LIN {X 0,Y 466.003,Z 780.81,A -85,B 0,C 180,E1 14179.349,E2 14179.349} C_VEL
LIN {X 0,Y 466.055,Z 780.81,A -85,B 0,C 180,E1 14186.554,E2 14186.554} C_VEL
LIN {X 0,Y 466.342,Z 780.81,A -85,B 0,C 180,E1 14193.024,E2 14193.024} C_VEL
LIN {X 0,Y 466.575,Z 780.81,A -85,B 0,C 180,E1 14199.925,E2 14199.925} C_VEL
LIN {X 0,Y 466.793,Z 780.81,A -85,B 0,C 180,E1 14206.211,E2 14206.211} C_VEL
LIN {X 0,Y 467.178,Z 780.81,A -85,B 0,C 180,E1 14212.565,E2 14212.565} C_VEL
LIN {X 0,Y 467.507,Z 780.81,A -85,B 0,C 180,E1 14218.145,E2 14218.145} C_VEL
LIN {X 0,Y 467.363,Z 780.81,A -85,B 0,C 180,E1 14223.704,E2 14223.704} C_VEL
LIN {X 0,Y 467.109,Z 780.81,A -85,B 0,C 180,E1 14229.304,E2 14229.304} C_VEL
LIN {X 0,Y 466.805,Z 780.81,A -85,B 0,C 180,E1 14235.003,E2 14235.003} C_VEL
LIN {X 0,Y 466.56,Z 780.81,A -85,B 0,C 180,E1 14240.865,E2 14240.865} C_VEL
LIN {X 0,Y 466.356,Z 780.81,A -85,B 0,C 180,E1 14246.969,E2 14246.969} C_VEL
LIN {X 0,Y 466.141,Z 780.81,A -85,B 0,C 180,E1 14253.432,E2 14253.432} C_VEL
LIN {X 0,Y 466.096,Z 780.943,A -85,B 0,C 180,E1 14257.269,E2 14257.269} C_VEL
LIN {X 0,Y 468.35,Z 786.358,A -85,B 0,C 180,E1 14257.738,E2 14257.738} C_VEL
LIN {X 0,Y 490.215,Z 820.764,A -85,B 0,C 180,E1 14261.492,E2 14261.492} C_VEL
LIN {X 0,Y 509.708,Z 858.555,A -85,B 0,C 180,E1 14264.767,E2 14264.767} C_VEL
LIN {X 0,Y 518.237,Z 880.593,A -85,B 0,C 180,E1 14266.483,E2 14266.483} C_VEL
LIN {X 0,Y 512.004,Z 925.358,A -85,B 0,C 180,E1 14268.177,E2 14268.177} C_VEL
LIN {X 0,Y 504.346,Z 968.699,A -85,B 0,C 180,E1 14270.608,E2 14270.608} C_VEL
LIN {X 0,Y 495.859,Z 1008.879,A -85,B 0,C 180,E1 14273.729,E2 14273.729} C_VEL
LIN {X 0,Y 487.965,Z 1043.053,A -85,B 0,C 180,E1 14277.25,E2 14277.25} C_VEL
LIN {X 0,Y 480.836,Z 1073.807,A -85,B 0,C 180,E1 14281.363,E2 14281.363} C_VEL
LIN {X 0,Y 474.612,Z 1101.899,A -85,B 0,C 180,E1 14286.298,E2 14286.298} C_VEL
LIN {X 0,Y 470.527,Z 1124.762,A -85,B 0,C 180,E1 14291.751,E2 14291.751} C_VEL
LIN {X 0,Y 468.531,Z 1140.188,A -85,B 0,C 180,E1 14296.951,E2 14296.951} C_VEL
LIN {X 0,Y 467.871,Z 1149.631,A -85,B 0,C 180,E1 14301.642,E2 14301.642} C_VEL
LIN {X 0,Y 467.662,Z 1154.817,A -85,B 0,C 180,E1 14306.294,E2 14306.294} C_VEL
LIN {X 0,Y 467.72,Z 1156.159,A -85,B 0,C 180,E1 14309.999,E2 14309.999} C_VEL
LIN {X 0,Y 467.629,Z 1155.649,A -85,B 0,C 180,E1 14312.192,E2 14312.192} C_VEL
LIN {X 0,Y 463.625,Z 1154.407,A -85,B 0,C 180,E1 14314.275,E2 14314.275} C_VEL
LIN {X 0,Y 459.843,Z 1152.277,A -85,B 0,C 180,E1 14316.387,E2 14316.387} C_VEL
LIN {X 0,Y 460.346,Z 1144.47,A -85,B 0,C 180,E1 14321.358,E2 14321.358} C_VEL
LIN {X 0,Y 461.991,Z 1131.343,A -85,B 0,C 180,E1 14326.629,E2 14326.629} C_VEL
LIN {X 0,Y 465.491,Z 1111.513,A -85,B 0,C 180,E1 14332.135,E2 14332.135} C_VEL
LIN {X 0,Y 471.08,Z 1086.781,A -85,B 0,C 180,E1 14337.199,E2 14337.199} C_VEL
LIN {X 0,Y 478.526,Z 1057.544,A -85,B 0,C 180,E1 14341.738,E2 14341.738} C_VEL
LIN {X 0,Y 487.44,Z 1023.022,A -85,B 0,C 180,E1 14345.812,E2 14345.812} C_VEL
LIN {X 0,Y 497.158,Z 982.841,A -85,B 0,C 180,E1 14349.34,E2 14349.34} C_VEL
LIN {X 0,Y 506.149,Z 940.056,A -85,B 0,C 180,E1 14352.054,E2 14352.054} C_VEL
LIN {X 0,Y 513.496,Z 896.79,A -85,B 0,C 180,E1 14353.955,E2 14353.955} C_VEL
LIN {X 0,Y 514.956,Z 882.197,A -85,B 0,C 180,E1 14354.501,E2 14354.501} C_VEL
LIN {X 0,Y 499.256,Z 847.046,A -85,B 0,C 180,E1 14357.774,E2 14357.774} C_VEL
LIN {X 0,Y 478.485,Z 812.037,A -85,B 0,C 180,E1 14361.711,E2 14361.711} C_VEL
LIN {X 0,Y 464.229,Z 791.641,A -85,B 0,C 180,E1 14364.642,E2 14364.642} C_VEL
LIN {X 0,Y 461.04,Z 786.903,A -85,B 0,C 180,E1 14365.359,E2 14365.359} C_VEL
LIN {X 0,Y 458.257,Z 781.978,A -85,B 0,C 180,E1 14366.028,E2 14366.028} C_VEL
LIN {X 0,Y 458.165,Z 780.81,A -85,B 0,C 180,E1 14366.133,E2 14366.133} C_VEL
LIN {X 0,Y 458.415,Z 780.81,A -85,B 0,C 180,E1 14372.873,E2 14372.873} C_VEL
LIN {X 0,Y 458.576,Z 780.81,A -85,B 0,C 180,E1 14378.755,E2 14378.755} C_VEL
LIN {X 0,Y 458.834,Z 780.81,A -85,B 0,C 180,E1 14384.73,E2 14384.73} C_VEL
LIN {X 0,Y 459.194,Z 780.81,A -85,B 0,C 180,E1 14390.828,E2 14390.828} C_VEL
LIN {X 0,Y 459.536,Z 780.81,A -85,B 0,C 180,E1 14396.233,E2 14396.233} C_VEL
LIN {X 0,Y 459.624,Z 780.81,A -85,B 0,C 180,E1 14401.887,E2 14401.887} C_VEL
LIN {X 0,Y 459.276,Z 780.81,A -85,B 0,C 180,E1 14407.564,E2 14407.564} C_VEL
LIN {X 0,Y 459.011,Z 780.81,A -85,B 0,C 180,E1 14413.324,E2 14413.324} C_VEL
LIN {X 0,Y 458.683,Z 780.81,A -85,B 0,C 180,E1 14419.235,E2 14419.235} C_VEL
LIN {X 0,Y 458.385,Z 780.81,A -85,B 0,C 180,E1 14425.374,E2 14425.374} C_VEL
LIN {X 0,Y 458.219,Z 780.81,A -85,B 0,C 180,E1 14431.37,E2 14431.37} C_VEL
LIN {X 0,Y 460.406,Z 786.283,A -85,B 0,C 180,E1 14431.966,E2 14431.966} C_VEL
LIN {X 0,Y 463.2,Z 789.773,A -85,B 0,C 180,E1 14432.582,E2 14432.582} C_VEL
LIN {X 0,Y 482.614,Z 818.941,A -85,B 0,C 180,E1 14436.642,E2 14436.642} C_VEL
LIN {X 0,Y 500.16,Z 852.088,A -85,B 0,C 180,E1 14440.434,E2 14440.434} C_VEL
LIN {X 0,Y 512.562,Z 884.16,A -85,B 0,C 180,E1 14443.642,E2 14443.642} C_VEL
LIN {X 0,Y 504.897,Z 927.615,A -85,B 0,C 180,E1 14445.867,E2 14445.867} C_VEL
LIN {X 0,Y 496.016,Z 968.133,A -85,B 0,C 180,E1 14448.793,E2 14448.793} C_VEL
LIN {X 0,Y 486.772,Z 1004.454,A -85,B 0,C 180,E1 14452.331,E2 14452.331} C_VEL
LIN {X 0,Y 478.378,Z 1035.552,A -85,B 0,C 180,E1 14456.331,E2 14456.331} C_VEL
LIN {X 0,Y 471.191,Z 1062.29,A -85,B 0,C 180,E1 14460.815,E2 14460.815} C_VEL
LIN {X 0,Y 465.51,Z 1085.609,A -85,B 0,C 180,E1 14466.062,E2 14466.062} C_VEL
LIN {X 0,Y 462.178,Z 1102.875,A -85,B 0,C 180,E1 14471.451,E2 14471.451} C_VEL
LIN {X 0,Y 460.451,Z 1114.458,A -85,B 0,C 180,E1 14476.72,E2 14476.72} C_VEL
LIN {X 0,Y 459.92,Z 1119.813,A -85,B 0,C 180,E1 14480.546,E2 14480.546} C_VEL
LIN {X 0,Y 459.641,Z 1123.056,A -85,B 0,C 180,E1 14486.231,E2 14486.231} C_VEL
LIN {X 0,Y 459.933,Z 1120.944,A -85,B 0,C 180,E1 14491.884,E2 14491.884} C_VEL
LIN {X 0,Y 460.385,Z 1115.045,A -85,B 0,C 180,E1 14496.598,E2 14496.598} C_VEL
LIN {X 0,Y 461.817,Z 1103.979,A -85,B 0,C 180,E1 14501.802,E2 14501.802} C_VEL
LIN {X 0,Y 464.72,Z 1087.594,A -85,B 0,C 180,E1 14507.018,E2 14507.018} C_VEL
LIN {X 0,Y 469.803,Z 1064.997,A -85,B 0,C 180,E1 14512.207,E2 14512.207} C_VEL
LIN {X 0,Y 476.391,Z 1038.632,A -85,B 0,C 180,E1 14516.752,E2 14516.752} C_VEL
LIN {X 0,Y 484.526,Z 1006.922,A -85,B 0,C 180,E1 14520.912,E2 14520.912} C_VEL
LIN {X 0,Y 493.645,Z 968.867,A -85,B 0,C 180,E1 14524.653,E2 14524.653} C_VEL
LIN {X 0,Y 502.271,Z 927.064,A -85,B 0,C 180,E1 14527.671,E2 14527.671} C_VEL
LIN {X 0,Y 509.568,Z 883.42,A -85,B 0,C 180,E1 14529.892,E2 14529.892} C_VEL
LIN {X 0,Y 495.699,Z 847.197,A -85,B 0,C 180,E1 14533.224,E2 14533.224} C_VEL
LIN {X 0,Y 476.674,Z 811.093,A -85,B 0,C 180,E1 14536.915,E2 14536.915} C_VEL
LIN {X 0,Y 460.205,Z 786.237,A -85,B 0,C 180,E1 14539.979,E2 14539.979} C_VEL
LIN {X 0,Y 458.009,Z 780.81,A -85,B 0,C 180,E1 14540.535,E2 14540.535} C_VEL
LIN {X 0,Y 458.055,Z 780.81,A -85,B 0,C 180,E1 14545.89,E2 14545.89} C_VEL
LIN {X 0,Y 458.379,Z 780.81,A -85,B 0,C 180,E1 14552.516,E2 14552.516} C_VEL
LIN {X 0,Y 458.588,Z 780.81,A -85,B 0,C 180,E1 14558.749,E2 14558.749} C_VEL
LIN {X 0,Y 458.832,Z 780.81,A -85,B 0,C 180,E1 14564.724,E2 14564.724} C_VEL
LIN {X 0,Y 459.215,Z 780.81,A -85,B 0,C 180,E1 14570.825,E2 14570.825} C_VEL
LIN {X 0,Y 459.558,Z 780.81,A -85,B 0,C 180,E1 14576.227,E2 14576.227} C_VEL
LIN {X 0,Y 459.639,Z 780.81,A -85,B 0,C 180,E1 14581.881,E2 14581.881} C_VEL
LIN {X 0,Y 459.248,Z 780.81,A -85,B 0,C 180,E1 14587.559,E2 14587.559} C_VEL
LIN {X 0,Y 458.996,Z 780.81,A -85,B 0,C 180,E1 14593.319,E2 14593.319} C_VEL
LIN {X 0,Y 458.715,Z 780.81,A -85,B 0,C 180,E1 14599.227,E2 14599.227} C_VEL
LIN {X 0,Y 458.424,Z 780.81,A -85,B 0,C 180,E1 14605.366,E2 14605.366} C_VEL
LIN {X 0,Y 458.26,Z 780.81,A -85,B 0,C 180,E1 14611.834,E2 14611.834} C_VEL
LIN {X 0,Y 458.148,Z 781.129,A -85,B 0,C 180,E1 14616.023,E2 14616.023} C_VEL
LIN {X 0,Y 460.626,Z 786.52,A -85,B 0,C 180,E1 14616.555,E2 14616.555} C_VEL
LIN {X 0,Y 480.891,Z 818.052,A -85,B 0,C 180,E1 14620.229,E2 14620.229} C_VEL
LIN {X 0,Y 500.554,Z 854.498,A -85,B 0,C 180,E1 14623.632,E2 14623.632} C_VEL
LIN {X 0,Y 512.078,Z 882.629,A -85,B 0,C 180,E1 14625.954,E2 14625.954} C_VEL
LIN {X 0,Y 505.842,Z 925.769,A -85,B 0,C 180,E1 14627.621,E2 14627.621} C_VEL
LIN {X 0,Y 497.732,Z 969.89,A -85,B 0,C 180,E1 14630.137,E2 14630.137} C_VEL
LIN {X 0,Y 488.886,Z 1010.227,A -85,B 0,C 180,E1 14633.327,E2 14633.327} C_VEL
LIN {X 0,Y 480.144,Z 1046.596,A -85,B 0,C 180,E1 14637.199,E2 14637.199} C_VEL
LIN {X 0,Y 472.886,Z 1076.357,A -85,B 0,C 180,E1 14641.358,E2 14641.358} C_VEL
LIN {X 0,Y 466.88,Z 1102.629,A -85,B 0,C 180,E1 14646.134,E2 14646.134} C_VEL
LIN {X 0,Y 462.745,Z 1124.874,A -85,B 0,C 180,E1 14651.571,E2 14651.571} C_VEL
LIN {X 0,Y 460.587,Z 1141.036,A -85,B 0,C 180,E1 14657.204,E2 14657.204} C_VEL
LIN {X 0,Y 459.892,Z 1150.634,A -85,B 0,C 180,E1 14662.447,E2 14662.447} C_VEL
LIN {X 0,Y 459.836,Z 1155.529,A -85,B 0,C 180,E1 14668.116,E2 14668.116} C_VEL
LIN {X 0,Y 459.733,Z 1155.398,A -85,B 0,C 180,E1 14672.175,E2 14672.175} C_VEL
LIN {X 0,Y 459.843,Z 1152.277,A -85,B 0,C 180,E1 14676.387,E2 14676.387} C_VEL
LIN {X 0,Y 457.472,Z 1150.386,A -85,B 0,C 180,E1 14677.982,E2 14677.982} C_VEL
LIN {X 0,Y 452.366,Z 1146.556,A -85,B 0,C 180,E1 14680.355,E2 14680.355} C_VEL
LIN {X 0,Y 452.306,Z 1146.036,A -85,B 0,C 180,E1 14680.627,E2 14680.627} C_VEL
LIN {X 0,Y 453.777,Z 1133.828,A -85,B 0,C 180,E1 14685.945,E2 14685.945} C_VEL
LIN {X 0,Y 456.962,Z 1116.098,A -85,B 0,C 180,E1 14691.33,E2 14691.33} C_VEL
LIN {X 0,Y 462.798,Z 1090.841,A -85,B 0,C 180,E1 14696.893,E2 14696.893} C_VEL
LIN {X 0,Y 470.93,Z 1060.042,A -85,B 0,C 180,E1 14701.903,E2 14701.903} C_VEL
LIN {X 0,Y 480.579,Z 1024.039,A -85,B 0,C 180,E1 14706.264,E2 14706.264} C_VEL
LIN {X 0,Y 490.627,Z 984.162,A -85,B 0,C 180,E1 14709.83,E2 14709.83} C_VEL
LIN {X 0,Y 499.865,Z 941.995,A -85,B 0,C 180,E1 14712.562,E2 14712.562} C_VEL
LIN {X 0,Y 507.349,Z 900.29,A -85,B 0,C 180,E1 14714.452,E2 14714.452} C_VEL
LIN {X 0,Y 508.891,Z 884.922,A -85,B 0,C 180,E1 14715.065,E2 14715.065} C_VEL
LIN {X 0,Y 493.722,Z 850.498,A -85,B 0,C 180,E1 14718.391,E2 14718.391} C_VEL
LIN {X 0,Y 474.535,Z 817.647,A -85,B 0,C 180,E1 14722.205,E2 14722.205} C_VEL
LIN {X 0,Y 457.343,Z 792.903,A -85,B 0,C 180,E1 14725.895,E2 14725.895} C_VEL
LIN {X 0,Y 453.216,Z 786.958,A -85,B 0,C 180,E1 14726.882,E2 14726.882} C_VEL
LIN {X 0,Y 450.415,Z 782.207,A -85,B 0,C 180,E1 14727.6,E2 14727.6} C_VEL
LIN {X 0,Y 450.283,Z 780.81,A -85,B 0,C 180,E1 14727.756,E2 14727.756} C_VEL
LIN {X 0,Y 450.496,Z 780.81,A -85,B 0,C 180,E1 14734.155,E2 14734.155} C_VEL
LIN {X 0,Y 450.716,Z 780.81,A -85,B 0,C 180,E1 14740.418,E2 14740.418} C_VEL
LIN {X 0,Y 451.016,Z 780.81,A -85,B 0,C 180,E1 14746.441,E2 14746.441} C_VEL
LIN {X 0,Y 451.316,Z 780.81,A -85,B 0,C 180,E1 14752.308,E2 14752.308} C_VEL
LIN {X 0,Y 451.682,Z 780.81,A -85,B 0,C 180,E1 14758.086,E2 14758.086} C_VEL
LIN {X 0,Y 451.543,Z 780.81,A -85,B 0,C 180,E1 14763.84,E2 14763.84} C_VEL
LIN {X 0,Y 451.271,Z 780.81,A -85,B 0,C 180,E1 14769.64,E2 14769.64} C_VEL
LIN {X 0,Y 450.963,Z 780.81,A -85,B 0,C 180,E1 14775.55,E2 14775.55} C_VEL
LIN {X 0,Y 450.632,Z 780.81,A -85,B 0,C 180,E1 14781.645,E2 14781.645} C_VEL
LIN {X 0,Y 450.369,Z 780.81,A -85,B 0,C 180,E1 14788.015,E2 14788.015} C_VEL
LIN {X 0,Y 450.369,Z 781.276,A -85,B 0,C 180,E1 14789.825,E2 14789.825} C_VEL
LIN {X 0,Y 452.709,Z 786.471,A -85,B 0,C 180,E1 14790.463,E2 14790.463} C_VEL
LIN {X 0,Y 455.413,Z 789.825,A -85,B 0,C 180,E1 14791.103,E2 14791.103} C_VEL
LIN {X 0,Y 472.547,Z 815.076,A -85,B 0,C 180,E1 14794.929,E2 14794.929} C_VEL
LIN {X 0,Y 489.417,Z 844.882,A -85,B 0,C 180,E1 14798.666,E2 14798.666} C_VEL
LIN {X 0,Y 503.111,Z 877.093,A -85,B 0,C 180,E1 14802.12,E2 14802.12} C_VEL
LIN {X 0,Y 506.394,Z 888.401,A -85,B 0,C 180,E1 14803.199,E2 14803.199} C_VEL
LIN {X 0,Y 498.875,Z 928.512,A -85,B 0,C 180,E1 14805.288,E2 14805.288} C_VEL
LIN {X 0,Y 489.595,Z 969.436,A -85,B 0,C 180,E1 14808.28,E2 14808.28} C_VEL
LIN {X 0,Y 479.894,Z 1006.088,A -85,B 0,C 180,E1 14811.917,E2 14811.917} C_VEL
LIN {X 0,Y 471.205,Z 1036.913,A -85,B 0,C 180,E1 14815.973,E2 14815.973} C_VEL
LIN {X 0,Y 463.985,Z 1062.615,A -85,B 0,C 180,E1 14820.363,E2 14820.363} C_VEL
LIN {X 0,Y 457.973,Z 1086.049,A -85,B 0,C 180,E1 14825.721,E2 14825.721} C_VEL
LIN {X 0,Y 454.402,Z 1103.478,A -85,B 0,C 180,E1 14831.279,E2 14831.279} C_VEL
LIN {X 0,Y 452.616,Z 1114.687,A -85,B 0,C 180,E1 14836.486,E2 14836.486} C_VEL
LIN {X 0,Y 451.835,Z 1121.751,A -85,B 0,C 180,E1 14842.313,E2 14842.313} C_VEL
LIN {X 0,Y 451.783,Z 1123.23,A -85,B 0,C 180,E1 14848.084,E2 14848.084} C_VEL
LIN {X 0,Y 452.171,Z 1119.382,A -85,B 0,C 180,E1 14853.833,E2 14853.833} C_VEL
LIN {X 0,Y 453.146,Z 1110.057,A -85,B 0,C 180,E1 14859.599,E2 14859.599} C_VEL
LIN {X 0,Y 455.801,Z 1094.608,A -85,B 0,C 180,E1 14865.381,E2 14865.381} C_VEL
LIN {X 0,Y 460.243,Z 1074.335,A -85,B 0,C 180,E1 14870.689,E2 14870.689} C_VEL
LIN {X 0,Y 466.4,Z 1050.103,A -85,B 0,C 180,E1 14875.424,E2 14875.424} C_VEL
LIN {X 0,Y 474.359,Z 1020.232,A -85,B 0,C 180,E1 14879.852,E2 14879.852} C_VEL
LIN {X 0,Y 483.758,Z 983.33,A -85,B 0,C 180,E1 14883.943,E2 14883.943} C_VEL
LIN {X 0,Y 493.261,Z 942.016,A -85,B 0,C 180,E1 14887.293,E2 14887.293} C_VEL
LIN {X 0,Y 501.024,Z 901.017,A -85,B 0,C 180,E1 14889.687,E2 14889.687} C_VEL
LIN {X 0,Y 503.111,Z 885.592,A -85,B 0,C 180,E1 14890.437,E2 14890.437} C_VEL
LIN {X 0,Y 489.101,Z 848.95,A -85,B 0,C 180,E1 14893.943,E2 14893.943} C_VEL
LIN {X 0,Y 471.255,Z 814.96,A -85,B 0,C 180,E1 14897.571,E2 14897.571} C_VEL
LIN {X 0,Y 452.843,Z 786.776,A -85,B 0,C 180,E1 14901.17,E2 14901.17} C_VEL
LIN {X 0,Y 450.18,Z 782.05,A -85,B 0,C 180,E1 14901.749,E2 14901.749} C_VEL
LIN {X 0,Y 450.107,Z 780.81,A -85,B 0,C 180,E1 14901.897,E2 14901.897} C_VEL
LIN {X 0,Y 450.174,Z 780.81,A -85,B 0,C 180,E1 14907.518,E2 14907.518} C_VEL
LIN {X 0,Y 450.47,Z 780.81,A -85,B 0,C 180,E1 14914.147,E2 14914.147} C_VEL
LIN {X 0,Y 450.728,Z 780.81,A -85,B 0,C 180,E1 14920.412,E2 14920.412} C_VEL
LIN {X 0,Y 451.015,Z 780.81,A -85,B 0,C 180,E1 14926.435,E2 14926.435} C_VEL
LIN {X 0,Y 451.327,Z 780.81,A -85,B 0,C 180,E1 14933.141,E2 14933.141} C_VEL
LIN {X 0,Y 451.713,Z 780.81,A -85,B 0,C 180,E1 14938.08,E2 14938.08} C_VEL
LIN {X 0,Y 451.541,Z 780.81,A -85,B 0,C 180,E1 14943.834,E2 14943.834} C_VEL
LIN {X 0,Y 451.26,Z 780.81,A -85,B 0,C 180,E1 14949.634,E2 14949.634} C_VEL
LIN {X 0,Y 450.932,Z 780.81,A -85,B 0,C 180,E1 14955.545,E2 14955.545} C_VEL
LIN {X 0,Y 450.661,Z 780.81,A -85,B 0,C 180,E1 14961.637,E2 14961.637} C_VEL
LIN {X 0,Y 450.406,Z 780.81,A -85,B 0,C 180,E1 14968.006,E2 14968.006} C_VEL
LIN {X 0,Y 450.224,Z 780.81,A -85,B 0,C 180,E1 14974.66,E2 14974.66} C_VEL
LIN {X 0,Y 452.498,Z 786.331,A -85,B 0,C 180,E1 14975.221,E2 14975.221} C_VEL
LIN {X 0,Y 468.108,Z 809.74,A -85,B 0,C 180,E1 14978.254,E2 14978.254} C_VEL
LIN {X 0,Y 488.269,Z 844.522,A -85,B 0,C 180,E1 14981.862,E2 14981.862} C_VEL
LIN {X 0,Y 504.735,Z 881.742,A -85,B 0,C 180,E1 14985.154,E2 14985.154} C_VEL
LIN {X 0,Y 505.776,Z 886.831,A -85,B 0,C 180,E1 14985.49,E2 14985.49} C_VEL
LIN {X 0,Y 499.132,Z 929.42,A -85,B 0,C 180,E1 14987.211,E2 14987.211} C_VEL
LIN {X 0,Y 491.175,Z 970.88,A -85,B 0,C 180,E1 14989.64,E2 14989.64} C_VEL
LIN {X 0,Y 482.094,Z 1010.81,A -85,B 0,C 180,E1 14992.848,E2 14992.848} C_VEL
LIN {X 0,Y 472.801,Z 1048.094,A -85,B 0,C 180,E1 14996.898,E2 14996.898} C_VEL
LIN {X 0,Y 464.517,Z 1080.856,A -85,B 0,C 180,E1 15001.671,E2 15001.671} C_VEL
LIN {X 0,Y 458.291,Z 1107.776,A -85,B 0,C 180,E1 15006.943,E2 15006.943} C_VEL
LIN {X 0,Y 454.536,Z 1127.489,A -85,B 0,C 180,E1 15012.173,E2 15012.173} C_VEL
LIN {X 0,Y 452.637,Z 1141.837,A -85,B 0,C 180,E1 15017.466,E2 15017.466} C_VEL
LIN {X 0,Y 452.023,Z 1150.33,A -85,B 0,C 180,E1 15022.314,E2 15022.314} C_VEL
LIN {X 0,Y 451.955,Z 1155.246,A -85,B 0,C 180,E1 15028.083,E2 15028.083} C_VEL
LIN {X 0,Y 451.902,Z 1155.269,A -85,B 0,C 180,E1 15031.915,E2 15031.915} C_VEL
LIN {X 0,Y 452.025,Z 1150.557,A -85,B 0,C 180,E1 15037.683,E2 15037.683} C_VEL
LIN {X 0,Y 452.306,Z 1146.036,A -85,B 0,C 180,E1 15040.627,E2 15040.627} C_VEL
LIN {X 0,Y 448.774,Z 1141.925,A -85,B 0,C 180,E1 15042.743,E2 15042.743} C_VEL
LIN {X 0,Y 445.465,Z 1137.142,A -85,B 0,C 180,E1 15044.878,E2 15044.878} C_VEL
LIN {X 0,Y 448.218,Z 1121.269,A -85,B 0,C 180,E1 15050.215,E2 15050.215} C_VEL
LIN {X 0,Y 453.373,Z 1098.991,A -85,B 0,C 180,E1 15055.675,E2 15055.675} C_VEL
LIN {X 0,Y 461.021,Z 1070.776,A -85,B 0,C 180,E1 15060.806,E2 15060.806} C_VEL
LIN {X 0,Y 470.809,Z 1035.517,A -85,B 0,C 180,E1 15065.572,E2 15065.572} C_VEL
LIN {X 0,Y 481.48,Z 996.197,A -85,B 0,C 180,E1 15069.466,E2 15069.466} C_VEL
LIN {X 0,Y 491.726,Z 953.378,A -85,B 0,C 180,E1 15072.536,E2 15072.536} C_VEL
LIN {X 0,Y 499.965,Z 911.064,A -85,B 0,C 180,E1 15074.671,E2 15074.671} C_VEL
LIN {X 0,Y 502.984,Z 887.991,A -85,B 0,C 180,E1 15075.613,E2 15075.613} C_VEL
LIN {X 0,Y 488.697,Z 854.787,A -85,B 0,C 180,E1 15078.931,E2 15078.931} C_VEL
LIN {X 0,Y 470.369,Z 822.869,A -85,B 0,C 180,E1 15082.755,E2 15082.755} C_VEL
LIN {X 0,Y 453.676,Z 798.649,A -85,B 0,C 180,E1 15086.449,E2 15086.449} C_VEL
LIN {X 0,Y 445.848,Z 787.309,A -85,B 0,C 180,E1 15088.421,E2 15088.421} C_VEL
LIN {X 0,Y 442.676,Z 782.833,A -85,B 0,C 180,E1 15089.271,E2 15089.271} C_VEL
LIN {X 0,Y 442.415,Z 780.81,A -85,B 0,C 180,E1 15089.433,E2 15089.433} C_VEL
LIN {X 0,Y 442.587,Z 780.81,A -85,B 0,C 180,E1 15095.821,E2 15095.821} C_VEL
LIN {X 0,Y 442.923,Z 780.81,A -85,B 0,C 180,E1 15102.794,E2 15102.794} C_VEL
LIN {X 0,Y 443.167,Z 780.81,A -85,B 0,C 180,E1 15108.2,E2 15108.2} C_VEL
LIN {X 0,Y 443.508,Z 780.81,A -85,B 0,C 180,E1 15114.137,E2 15114.137} C_VEL
LIN {X 0,Y 443.961,Z 780.81,A -85,B 0,C 180,E1 15120.003,E2 15120.003} C_VEL
LIN {X 0,Y 443.58,Z 780.81,A -85,B 0,C 180,E1 15125.868,E2 15125.868} C_VEL
LIN {X 0,Y 443.208,Z 780.81,A -85,B 0,C 180,E1 15131.805,E2 15131.805} C_VEL
LIN {X 0,Y 442.903,Z 780.81,A -85,B 0,C 180,E1 15137.882,E2 15137.882} C_VEL
LIN {X 0,Y 442.562,Z 780.81,A -85,B 0,C 180,E1 15144.187,E2 15144.187} C_VEL
LIN {X 0,Y 442.467,Z 780.935,A -85,B 0,C 180,E1 15148.083,E2 15148.083} C_VEL
LIN {X 0,Y 444.419,Z 786.044,A -85,B 0,C 180,E1 15148.687,E2 15148.687} C_VEL
LIN {X 0,Y 447.508,Z 789.498,A -85,B 0,C 180,E1 15149.469,E2 15149.469} C_VEL
LIN {X 0,Y 465.321,Z 815.546,A -85,B 0,C 180,E1 15153.715,E2 15153.715} C_VEL
LIN {X 0,Y 482.559,Z 845.746,A -85,B 0,C 180,E1 15157.721,E2 15157.721} C_VEL
LIN {X 0,Y 496.416,Z 878.028,A -85,B 0,C 180,E1 15161.345,E2 15161.345} C_VEL
LIN {X 0,Y 500.471,Z 890.799,A -85,B 0,C 180,E1 15162.652,E2 15162.652} C_VEL
LIN {X 0,Y 492.587,Z 930.897,A -85,B 0,C 180,E1 15164.792,E2 15164.792} C_VEL
LIN {X 0,Y 483.194,Z 970.718,A -85,B 0,C 180,E1 15167.755,E2 15167.755} C_VEL
LIN {X 0,Y 473.022,Z 1007.812,A -85,B 0,C 180,E1 15171.502,E2 15171.502} C_VEL
LIN {X 0,Y 463.69,Z 1039.531,A -85,B 0,C 180,E1 15175.796,E2 15175.796} C_VEL
LIN {X 0,Y 455.858,Z 1066.093,A -85,B 0,C 180,E1 15180.551,E2 15180.551} C_VEL
LIN {X 0,Y 450.004,Z 1088.196,A -85,B 0,C 180,E1 15185.847,E2 15185.847} C_VEL
LIN {X 0,Y 446.324,Z 1105.875,A -85,B 0,C 180,E1 15191.798,E2 15191.798} C_VEL
LIN {X 0,Y 444.603,Z 1116.444,A -85,B 0,C 180,E1 15197.238,E2 15197.238} C_VEL
LIN {X 0,Y 443.943,Z 1122.004,A -85,B 0,C 180,E1 15202.176,E2 15202.176} C_VEL
LIN {X 0,Y 443.883,Z 1123.517,A -85,B 0,C 180,E1 15208.05,E2 15208.05} C_VEL
LIN {X 0,Y 444.284,Z 1119.706,A -85,B 0,C 180,E1 15213.902,E2 15213.902} C_VEL
LIN {X 0,Y 445.315,Z 1110.413,A -85,B 0,C 180,E1 15219.77,E2 15219.77} C_VEL
LIN {X 0,Y 448.115,Z 1094.999,A -85,B 0,C 180,E1 15225.652,E2 15225.652} C_VEL
LIN {X 0,Y 452.757,Z 1074.82,A -85,B 0,C 180,E1 15231.035,E2 15231.035} C_VEL
LIN {X 0,Y 459.187,Z 1050.587,A -85,B 0,C 180,E1 15235.852,E2 15235.852} C_VEL
LIN {X 0,Y 467.467,Z 1020.757,A -85,B 0,C 180,E1 15240.338,E2 15240.338} C_VEL
LIN {X 0,Y 477.18,Z 984.027,A -85,B 0,C 180,E1 15244.463,E2 15244.463} C_VEL
LIN {X 0,Y 486.576,Z 944.764,A -85,B 0,C 180,E1 15247.702,E2 15247.702} C_VEL
LIN {X 0,Y 493.962,Z 907.657,A -85,B 0,C 180,E1 15249.974,E2 15249.974} C_VEL
LIN {X 0,Y 496.777,Z 888.196,A -85,B 0,C 180,E1 15250.961,E2 15250.961} C_VEL
LIN {X 0,Y 483.06,Z 851.902,A -85,B 0,C 180,E1 15254.556,E2 15254.556} C_VEL
LIN {X 0,Y 466.182,Z 819.137,A -85,B 0,C 180,E1 15258.182,E2 15258.182} C_VEL
LIN {X 0,Y 448.706,Z 792.411,A -85,B 0,C 180,E1 15261.73,E2 15261.73} C_VEL
LIN {X 0,Y 444.789,Z 786.672,A -85,B 0,C 180,E1 15262.578,E2 15262.578} C_VEL
LIN {X 0,Y 442.252,Z 781.808,A -85,B 0,C 180,E1 15263.176,E2 15263.176} C_VEL
LIN {X 0,Y 442.205,Z 780.81,A -85,B 0,C 180,E1 15263.319,E2 15263.319} C_VEL
LIN {X 0,Y 442.309,Z 780.81,A -85,B 0,C 180,E1 15269.175,E2 15269.175} C_VEL
LIN {X 0,Y 442.586,Z 780.81,A -85,B 0,C 180,E1 15275.814,E2 15275.814} C_VEL
LIN {X 0,Y 442.901,Z 780.81,A -85,B 0,C 180,E1 15282.118,E2 15282.118} C_VEL
LIN {X 0,Y 443.182,Z 780.81,A -85,B 0,C 180,E1 15288.194,E2 15288.194} C_VEL
LIN {X 0,Y 443.532,Z 780.81,A -85,B 0,C 180,E1 15294.132,E2 15294.132} C_VEL
LIN {X 0,Y 443.98,Z 780.81,A -85,B 0,C 180,E1 15299.997,E2 15299.997} C_VEL
LIN {X 0,Y 443.538,Z 780.81,A -85,B 0,C 180,E1 15305.862,E2 15305.862} C_VEL
LIN {X 0,Y 443.204,Z 780.81,A -85,B 0,C 180,E1 15311.799,E2 15311.799} C_VEL
LIN {X 0,Y 442.934,Z 780.81,A -85,B 0,C 180,E1 15317.875,E2 15317.875} C_VEL
LIN {X 0,Y 442.604,Z 780.81,A -85,B 0,C 180,E1 15324.178,E2 15324.178} C_VEL
LIN {X 0,Y 442.374,Z 780.81,A -85,B 0,C 180,E1 15330.813,E2 15330.813} C_VEL
LIN {X 0,Y 442.35,Z 780.81,A -85,B 0,C 180,E1 15333.247,E2 15333.247} C_VEL
LIN {X 0,Y 444.35,Z 786.05,A -85,B 0,C 180,E1 15333.786,E2 15333.786} C_VEL
LIN {X 0,Y 447.42,Z 790.27,A -85,B 0,C 180,E1 15334.449,E2 15334.449} C_VEL
LIN {X 0,Y 465.562,Z 817.63,A -85,B 0,C 180,E1 15338.064,E2 15338.064} C_VEL
LIN {X 0,Y 484.552,Z 851.858,A -85,B 0,C 180,E1 15341.641,E2 15341.641} C_VEL
LIN {X 0,Y 499.724,Z 887.726,A -85,B 0,C 180,E1 15344.887,E2 15344.887} C_VEL
LIN {X 0,Y 492.705,Z 931.993,A -85,B 0,C 180,E1 15346.742,E2 15346.742} C_VEL
LIN {X 0,Y 484.332,Z 973.317,A -85,B 0,C 180,E1 15349.234,E2 15349.234} C_VEL
LIN {X 0,Y 475.222,Z 1011.806,A -85,B 0,C 180,E1 15352.4,E2 15352.4} C_VEL
LIN {X 0,Y 465.618,Z 1048.934,A -85,B 0,C 180,E1 15356.514,E2 15356.514} C_VEL
LIN {X 0,Y 457.162,Z 1081.083,A -85,B 0,C 180,E1 15361.29,E2 15361.29} C_VEL
LIN {X 0,Y 450.584,Z 1108.152,A -85,B 0,C 180,E1 15366.704,E2 15366.704} C_VEL
LIN {X 0,Y 446.594,Z 1128.447,A -85,B 0,C 180,E1 15372.269,E2 15372.269} C_VEL
LIN {X 0,Y 444.809,Z 1141.515,A -85,B 0,C 180,E1 15377.242,E2 15377.242} C_VEL
LIN {X 0,Y 444.069,Z 1151.264,A -85,B 0,C 180,E1 15383.159,E2 15383.159} C_VEL
LIN {X 0,Y 444.051,Z 1154.961,A -85,B 0,C 180,E1 15388.049,E2 15388.049} C_VEL
LIN {X 0,Y 443.999,Z 1154.99,A -85,B 0,C 180,E1 15391.949,E2 15391.949} C_VEL
LIN {X 0,Y 444.13,Z 1150.296,A -85,B 0,C 180,E1 15397.821,E2 15397.821} C_VEL
LIN {X 0,Y 444.981,Z 1140.979,A -85,B 0,C 180,E1 15403.25,E2 15403.25} C_VEL
LIN {X 0,Y 445.465,Z 1137.142,A -85,B 0,C 180,E1 15404.878,E2 15404.878} C_VEL
LIN {X 0,Y 442.362,Z 1131.857,A -85,B 0,C 180,E1 15406.999,E2 15406.999} C_VEL
LIN {X 0,Y 439.532,Z 1125.859,A -85,B 0,C 180,E1 15409.118,E2 15409.118} C_VEL
LIN {X 0,Y 444.214,Z 1105.502,A -85,B 0,C 180,E1 15414.626,E2 15414.626} C_VEL
LIN {X 0,Y 451.375,Z 1079.396,A -85,B 0,C 180,E1 15419.872,E2 15419.872} C_VEL
LIN {X 0,Y 460.968,Z 1046.798,A -85,B 0,C 180,E1 15424.746,E2 15424.746} C_VEL
LIN {X 0,Y 471.508,Z 1010.098,A -85,B 0,C 180,E1 15428.824,E2 15428.824} C_VEL
LIN {X 0,Y 481.884,Z 970.383,A -85,B 0,C 180,E1 15432.062,E2 15432.062} C_VEL
LIN {X 0,Y 490.761,Z 929.924,A -85,B 0,C 180,E1 15434.465,E2 15434.465} C_VEL
LIN {X 0,Y 497.4,Z 891.915,A -85,B 0,C 180,E1 15436.084,E2 15436.084} C_VEL
LIN {X 0,Y 483.543,Z 859.018,A -85,B 0,C 180,E1 15439.484,E2 15439.484} C_VEL
LIN {X 0,Y 466.389,Z 828.472,A -85,B 0,C 180,E1 15443.256,E2 15443.256} C_VEL
LIN {X 0,Y 447.892,Z 800.867,A -85,B 0,C 180,E1 15447.566,E2 15447.566} C_VEL
LIN {X 0,Y 439.414,Z 788.588,A -85,B 0,C 180,E1 15449.838,E2 15449.838} C_VEL
LIN {X 0,Y 434.869,Z 783.135,A -85,B 0,C 180,E1 15451.126,E2 15451.126} C_VEL
LIN {X 0,Y 434.57,Z 780.81,A -85,B 0,C 180,E1 15451.48,E2 15451.48} C_VEL
LIN {X 0,Y 434.722,Z 780.81,A -85,B 0,C 180,E1 15457.527,E2 15457.527} C_VEL
LIN {X 0,Y 435.032,Z 780.81,A -85,B 0,C 180,E1 15463.872,E2 15463.872} C_VEL
LIN {X 0,Y 435.381,Z 780.81,A -85,B 0,C 180,E1 15470.011,E2 15470.011} C_VEL
LIN {X 0,Y 435.797,Z 780.81,A -85,B 0,C 180,E1 15476.027,E2 15476.027} C_VEL
LIN {X 0,Y 435.928,Z 780.81,A -85,B 0,C 180,E1 15481.989,E2 15481.989} C_VEL
LIN {X 0,Y 435.526,Z 780.81,A -85,B 0,C 180,E1 15487.979,E2 15487.979} C_VEL
LIN {X 0,Y 435.226,Z 780.81,A -85,B 0,C 180,E1 15494.067,E2 15494.067} C_VEL
LIN {X 0,Y 434.854,Z 780.81,A -85,B 0,C 180,E1 15500.334,E2 15500.334} C_VEL
LIN {X 0,Y 434.575,Z 781.116,A -85,B 0,C 180,E1 15506.192,E2 15506.192} C_VEL
LIN {X 0,Y 436.782,Z 786.334,A -85,B 0,C 180,E1 15506.919,E2 15506.919} C_VEL
LIN {X 0,Y 439.878,Z 789.739,A -85,B 0,C 180,E1 15507.771,E2 15507.771} C_VEL
LIN {X 0,Y 457.198,Z 814.438,A -85,B 0,C 180,E1 15512.203,E2 15512.203} C_VEL
LIN {X 0,Y 474.638,Z 844.613,A -85,B 0,C 180,E1 15516.469,E2 15516.469} C_VEL
LIN {X 0,Y 488.259,Z 875.049,A -85,B 0,C 180,E1 15520.107,E2 15520.107} C_VEL
LIN {X 0,Y 494.323,Z 895.032,A -85,B 0,C 180,E1 15522.179,E2 15522.179} C_VEL
LIN {X 0,Y 485.749,Z 936.005,A -85,B 0,C 180,E1 15524.466,E2 15524.466} C_VEL
LIN {X 0,Y 476.414,Z 973.48,A -85,B 0,C 180,E1 15527.354,E2 15527.354} C_VEL
LIN {X 0,Y 466.183,Z 1009.431,A -85,B 0,C 180,E1 15531.065,E2 15531.065} C_VEL
LIN {X 0,Y 456.006,Z 1042.785,A -85,B 0,C 180,E1 15535.714,E2 15535.714} C_VEL
LIN {X 0,Y 447.395,Z 1071.042,A -85,B 0,C 180,E1 15541.062,E2 15541.062} C_VEL
LIN {X 0,Y 441.727,Z 1091.525,A -85,B 0,C 180,E1 15546.354,E2 15546.354} C_VEL
LIN {X 0,Y 438.418,Z 1107.102,A -85,B 0,C 180,E1 15551.93,E2 15551.93} C_VEL
LIN {X 0,Y 436.754,Z 1116.675,A -85,B 0,C 180,E1 15557.005,E2 15557.005} C_VEL
LIN {X 0,Y 436.06,Z 1122.256,A -85,B 0,C 180,E1 15562.033,E2 15562.033} C_VEL
LIN {X 0,Y 435.987,Z 1123.804,A -85,B 0,C 180,E1 15568.015,E2 15568.015} C_VEL
LIN {X 0,Y 436.267,Z 1121.879,A -85,B 0,C 180,E1 15571.986,E2 15571.986} C_VEL
LIN {X 0,Y 436.813,Z 1116.057,A -85,B 0,C 180,E1 15576.955,E2 15576.955} C_VEL
LIN {X 0,Y 438.449,Z 1105.113,A -85,B 0,C 180,E1 15582.44,E2 15582.44} C_VEL
LIN {X 0,Y 442.244,Z 1087.109,A -85,B 0,C 180,E1 15588.426,E2 15588.426} C_VEL
LIN {X 0,Y 448.688,Z 1062.742,A -85,B 0,C 180,E1 15594.124,E2 15594.124} C_VEL
LIN {X 0,Y 457.285,Z 1032.828,A -85,B 0,C 180,E1 15599.227,E2 15599.227} C_VEL
LIN {X 0,Y 467.034,Z 998.148,A -85,B 0,C 180,E1 15603.612,E2 15603.612} C_VEL
LIN {X 0,Y 476.533,Z 961.539,A -85,B 0,C 180,E1 15607.05,E2 15607.05} C_VEL
LIN {X 0,Y 484.874,Z 923.858,A -85,B 0,C 180,E1 15609.71,E2 15609.71} C_VEL
LIN {X 0,Y 490.652,Z 891.43,A -85,B 0,C 180,E1 15611.44,E2 15611.44} C_VEL
LIN {X 0,Y 477.132,Z 854.846,A -85,B 0,C 180,E1 15615.171,E2 15615.171} C_VEL
LIN {X 0,Y 460.554,Z 822.306,A -85,B 0,C 180,E1 15618.911,E2 15618.911} C_VEL
LIN {X 0,Y 441.647,Z 793.271,A -85,B 0,C 180,E1 15622.97,E2 15622.97} C_VEL
LIN {X 0,Y 436.832,Z 786.608,A -85,B 0,C 180,E1 15624.07,E2 15624.07} C_VEL
LIN {X 0,Y 434.339,Z 781.366,A -85,B 0,C 180,E1 15624.714,E2 15624.714} C_VEL
LIN {X 0,Y 434.449,Z 780.81,A -85,B 0,C 180,E1 15630.862,E2 15630.862} C_VEL
LIN {X 0,Y 434.731,Z 780.81,A -85,B 0,C 180,E1 15637.521,E2 15637.521} C_VEL
LIN {X 0,Y 435.036,Z 780.81,A -85,B 0,C 180,E1 15643.866,E2 15643.866} C_VEL
LIN {X 0,Y 435.371,Z 780.81,A -85,B 0,C 180,E1 15650.005,E2 15650.005} C_VEL
LIN {X 0,Y 435.819,Z 780.81,A -85,B 0,C 180,E1 15656.021,E2 15656.021} C_VEL
LIN {X 0,Y 435.941,Z 780.81,A -85,B 0,C 180,E1 15661.983,E2 15661.983} C_VEL
LIN {X 0,Y 435.506,Z 780.81,A -85,B 0,C 180,E1 15667.973,E2 15667.973} C_VEL
LIN {X 0,Y 435.206,Z 780.81,A -85,B 0,C 180,E1 15674.061,E2 15674.061} C_VEL
LIN {X 0,Y 434.866,Z 780.81,A -85,B 0,C 180,E1 15680.327,E2 15680.327} C_VEL
LIN {X 0,Y 434.608,Z 780.81,A -85,B 0,C 180,E1 15686.864,E2 15686.864} C_VEL
LIN {X 0,Y 434.421,Z 780.81,A -85,B 0,C 180,E1 15691.711,E2 15691.711} C_VEL
LIN {X 0,Y 436.661,Z 786.339,A -85,B 0,C 180,E1 15692.349,E2 15692.349} C_VEL
LIN {X 0,Y 439.422,Z 789.852,A -85,B 0,C 180,E1 15692.979,E2 15692.979} C_VEL
LIN {X 0,Y 458.81,Z 818.948,A -85,B 0,C 180,E1 15697.068,E2 15697.068} C_VEL
LIN {X 0,Y 477.692,Z 852.639,A -85,B 0,C 180,E1 15700.788,E2 15700.788} C_VEL
LIN {X 0,Y 492.696,Z 888.032,A -85,B 0,C 180,E1 15704.128,E2 15704.128} C_VEL
LIN {X 0,Y 493.324,Z 893.32,A -85,B 0,C 180,E1 15704.467,E2 15704.467} C_VEL
LIN {X 0,Y 485.859,Z 937.07,A -85,B 0,C 180,E1 15706.387,E2 15706.387} C_VEL
LIN {X 0,Y 476.385,Z 980.586,A -85,B 0,C 180,E1 15709.166,E2 15709.166} C_VEL
LIN {X 0,Y 466.591,Z 1019.273,A -85,B 0,C 180,E1 15712.582,E2 15712.582} C_VEL
LIN {X 0,Y 457.787,Z 1052.053,A -85,B 0,C 180,E1 15716.433,E2 15716.433} C_VEL
LIN {X 0,Y 449.432,Z 1082.655,A -85,B 0,C 180,E1 15721.145,E2 15721.145} C_VEL
LIN {X 0,Y 442.748,Z 1109.294,A -85,B 0,C 180,E1 15726.648,E2 15726.648} C_VEL
LIN {X 0,Y 438.634,Z 1129.666,A -85,B 0,C 180,E1 15732.455,E2 15732.455} C_VEL
LIN {X 0,Y 436.705,Z 1143.166,A -85,B 0,C 180,E1 15738.016,E2 15738.016} C_VEL
LIN {X 0,Y 436.179,Z 1150.958,A -85,B 0,C 180,E1 15743.034,E2 15743.034} C_VEL
LIN {X 0,Y 436.165,Z 1154.677,A -85,B 0,C 180,E1 15748.013,E2 15748.013} C_VEL
LIN {X 0,Y 436.119,Z 1154.713,A -85,B 0,C 180,E1 15751.984,E2 15751.984} C_VEL
LIN {X 0,Y 436.244,Z 1150.035,A -85,B 0,C 180,E1 15757.963,E2 15757.963} C_VEL
LIN {X 0,Y 437.14,Z 1140.738,A -85,B 0,C 180,E1 15763.492,E2 15763.492} C_VEL
LIN {X 0,Y 439.532,Z 1125.859,A -85,B 0,C 180,E1 15769.118,E2 15769.118} C_VEL
LIN {X 0,Y 437.111,Z 1119.432,A -85,B 0,C 180,E1 15771.229,E2 15771.229} C_VEL
LIN {X 0,Y 434.967,Z 1112.329,A -85,B 0,C 180,E1 15773.326,E2 15773.326} C_VEL
LIN {X 0,Y 441.414,Z 1088.748,A -85,B 0,C 180,E1 15778.636,E2 15778.636} C_VEL
LIN {X 0,Y 450.461,Z 1059.224,A -85,B 0,C 180,E1 15783.606,E2 15783.606} C_VEL
LIN {X 0,Y 461.212,Z 1023.677,A -85,B 0,C 180,E1 15788.06,E2 15788.06} C_VEL
LIN {X 0,Y 471.878,Z 985.818,A -85,B 0,C 180,E1 15791.562,E2 15791.562} C_VEL
LIN {X 0,Y 481.674,Z 945.985,A -85,B 0,C 180,E1 15794.267,E2 15794.267} C_VEL
LIN {X 0,Y 490.114,Z 904.538,A -85,B 0,C 180,E1 15796.261,E2 15796.261} C_VEL
LIN {X 0,Y 491.354,Z 894.491,A -85,B 0,C 180,E1 15796.687,E2 15796.687} C_VEL
LIN {X 0,Y 477.505,Z 861.28,A -85,B 0,C 180,E1 15800.261,E2 15800.261} C_VEL
LIN {X 0,Y 460.408,Z 830.722,A -85,B 0,C 180,E1 15804.234,E2 15804.234} C_VEL
LIN {X 0,Y 443.768,Z 806.155,A -85,B 0,C 180,E1 15808.288,E2 15808.288} C_VEL
LIN {X 0,Y 434.688,Z 793.661,A -85,B 0,C 180,E1 15810.806,E2 15810.806} C_VEL
LIN {X 0,Y 430.351,Z 787.517,A -85,B 0,C 180,E1 15812.133,E2 15812.133} C_VEL
LIN {X 0,Y 426.89,Z 782.585,A -85,B 0,C 180,E1 15813.259,E2 15813.259} C_VEL
LIN {X 0,Y 426.668,Z 780.81,A -85,B 0,C 180,E1 15813.394,E2 15813.394} C_VEL
LIN {X 0,Y 426.875,Z 780.81,A -85,B 0,C 180,E1 15819.275,E2 15819.275} C_VEL
LIN {X 0,Y 427.219,Z 780.81,A -85,B 0,C 180,E1 15825.67,E2 15825.67} C_VEL
LIN {X 0,Y 427.567,Z 780.81,A -85,B 0,C 180,E1 15831.878,E2 15831.878} C_VEL
LIN {X 0,Y 427.987,Z 780.81,A -85,B 0,C 180,E1 15837.98,E2 15837.98} C_VEL
LIN {X 0,Y 427.808,Z 780.81,A -85,B 0,C 180,E1 15844.053,E2 15844.053} C_VEL
LIN {X 0,Y 427.505,Z 780.81,A -85,B 0,C 180,E1 15850.181,E2 15850.181} C_VEL
LIN {X 0,Y 427.074,Z 780.81,A -85,B 0,C 180,E1 15857.193,E2 15857.193} C_VEL
LIN {X 0,Y 426.671,Z 780.81,A -85,B 0,C 180,E1 15864.032,E2 15864.032} C_VEL
LIN {X 0,Y 428.829,Z 786.228,A -85,B 0,C 180,E1 15864.874,E2 15864.874} C_VEL
LIN {X 0,Y 432.063,Z 789.598,A -85,B 0,C 180,E1 15865.851,E2 15865.851} C_VEL
LIN {X 0,Y 446.797,Z 810.422,A -85,B 0,C 180,E1 15869.992,E2 15869.992} C_VEL
LIN {X 0,Y 463.265,Z 836.729,A -85,B 0,C 180,E1 15874.206,E2 15874.206} C_VEL
LIN {X 0,Y 478.504,Z 868.175,A -85,B 0,C 180,E1 15878.315,E2 15878.315} C_VEL
LIN {X 0,Y 488.361,Z 896.011,A -85,B 0,C 180,E1 15881.493,E2 15881.493} C_VEL
LIN {X 0,Y 479.5,Z 938.547,A -85,B 0,C 180,E1 15883.957,E2 15883.957} C_VEL
LIN {X 0,Y 469.931,Z 975.33,A -85,B 0,C 180,E1 15886.859,E2 15886.859} C_VEL
LIN {X 0,Y 459.351,Z 1011.012,A -85,B 0,C 180,E1 15890.62,E2 15890.62} C_VEL
LIN {X 0,Y 449.231,Z 1042.862,A -85,B 0,C 180,E1 15895.123,E2 15895.123} C_VEL
LIN {X 0,Y 440.342,Z 1070.703,A -85,B 0,C 180,E1 15900.444,E2 15900.444} C_VEL
LIN {X 0,Y 434.274,Z 1091.524,A -85,B 0,C 180,E1 15905.868,E2 15905.868} C_VEL
LIN {X 0,Y 430.691,Z 1107.31,A -85,B 0,C 180,E1 15911.594,E2 15911.594} C_VEL
LIN {X 0,Y 428.69,Z 1118.423,A -85,B 0,C 180,E1 15917.791,E2 15917.791} C_VEL
LIN {X 0,Y 428.04,Z 1123.632,A -85,B 0,C 180,E1 15923.922,E2 15923.922} C_VEL
LIN {X 0,Y 428.265,Z 1123.433,A -85,B 0,C 180,E1 15930.001,E2 15930.001} C_VEL
LIN {X 0,Y 428.735,Z 1117.913,A -85,B 0,C 180,E1 15936.071,E2 15936.071} C_VEL
LIN {X 0,Y 430.503,Z 1106.693,A -85,B 0,C 180,E1 15942.159,E2 15942.159} C_VEL
LIN {X 0,Y 433.836,Z 1090.9,A -85,B 0,C 180,E1 15947.746,E2 15947.746} C_VEL
LIN {X 0,Y 439.373,Z 1070.306,A -85,B 0,C 180,E1 15953.031,E2 15953.031} C_VEL
LIN {X 0,Y 447.399,Z 1043.005,A -85,B 0,C 180,E1 15958.221,E2 15958.221} C_VEL
LIN {X 0,Y 457.64,Z 1008.705,A -85,B 0,C 180,E1 15963.014,E2 15963.014} C_VEL
LIN {X 0,Y 468.226,Z 970.34,A -85,B 0,C 180,E1 15966.949,E2 15966.949} C_VEL
LIN {X 0,Y 478.088,Z 928.283,A -85,B 0,C 180,E1 15970.092,E2 15970.092} C_VEL
LIN {X 0,Y 484.35,Z 893.97,A -85,B 0,C 180,E1 15972,E2 15972} C_VEL
LIN {X 0,Y 471.578,Z 858.701,A -85,B 0,C 180,E1 15975.71,E2 15975.71} C_VEL
LIN {X 0,Y 455.863,Z 827.334,A -85,B 0,C 180,E1 15979.449,E2 15979.449} C_VEL
LIN {X 0,Y 438.43,Z 799.774,A -85,B 0,C 180,E1 15983.389,E2 15983.389} C_VEL
LIN {X 0,Y 429.462,Z 787.042,A -85,B 0,C 180,E1 15985.542,E2 15985.542} C_VEL
LIN {X 0,Y 426.568,Z 782.338,A -85,B 0,C 180,E1 15986.303,E2 15986.303} C_VEL
LIN {X 0,Y 426.422,Z 780.81,A -85,B 0,C 180,E1 15986.469,E2 15986.469} C_VEL
LIN {X 0,Y 426.585,Z 780.81,A -85,B 0,C 180,E1 15992.582,E2 15992.582} C_VEL
LIN {X 0,Y 426.897,Z 780.81,A -85,B 0,C 180,E1 15999.27,E2 15999.27} C_VEL
LIN {X 0,Y 427.216,Z 780.81,A -85,B 0,C 180,E1 16005.664,E2 16005.664} C_VEL
LIN {X 0,Y 427.591,Z 780.81,A -85,B 0,C 180,E1 16011.872,E2 16011.872} C_VEL
LIN {X 0,Y 428.015,Z 780.81,A -85,B 0,C 180,E1 16017.974,E2 16017.974} C_VEL
LIN {X 0,Y 427.801,Z 780.81,A -85,B 0,C 180,E1 16024.047,E2 16024.047} C_VEL
LIN {X 0,Y 427.5,Z 780.81,A -85,B 0,C 180,E1 16030.175,E2 16030.175} C_VEL
LIN {X 0,Y 427.063,Z 780.81,A -85,B 0,C 180,E1 16037.181,E2 16037.181} C_VEL
LIN {X 0,Y 426.759,Z 780.81,A -85,B 0,C 180,E1 16042.979,E2 16042.979} C_VEL
LIN {X 0,Y 426.514,Z 780.81,A -85,B 0,C 180,E1 16050.08,E2 16050.08} C_VEL
LIN {X 0,Y 428.54,Z 786.126,A -85,B 0,C 180,E1 16050.697,E2 16050.697} C_VEL
LIN {X 0,Y 431.52,Z 789.688,A -85,B 0,C 180,E1 16051.423,E2 16051.423} C_VEL
LIN {X 0,Y 449.675,Z 816.447,A -85,B 0,C 180,E1 16055.525,E2 16055.525} C_VEL
LIN {X 0,Y 469.057,Z 850.013,A -85,B 0,C 180,E1 16059.531,E2 16059.531} C_VEL
LIN {X 0,Y 484.611,Z 885.428,A -85,B 0,C 180,E1 16063.072,E2 16063.072} C_VEL
LIN {X 0,Y 487.307,Z 895.085,A -85,B 0,C 180,E1 16063.888,E2 16063.888} C_VEL
LIN {X 0,Y 479.576,Z 938.758,A -85,B 0,C 180,E1 16065.852,E2 16065.852} C_VEL
LIN {X 0,Y 469.966,Z 981.273,A -85,B 0,C 180,E1 16068.61,E2 16068.61} C_VEL
LIN {X 0,Y 459.524,Z 1021.002,A -85,B 0,C 180,E1 16072.189,E2 16072.189} C_VEL
LIN {X 0,Y 449.905,Z 1055.167,A -85,B 0,C 180,E1 16076.344,E2 16076.344} C_VEL
LIN {X 0,Y 441.56,Z 1084.654,A -85,B 0,C 180,E1 16081.081,E2 16081.081} C_VEL
LIN {X 0,Y 434.963,Z 1109.996,A -85,B 0,C 180,E1 16086.499,E2 16086.499} C_VEL
LIN {X 0,Y 430.881,Z 1129.312,A -85,B 0,C 180,E1 16092.128,E2 16092.128} C_VEL
LIN {X 0,Y 428.846,Z 1142.841,A -85,B 0,C 180,E1 16097.793,E2 16097.793} C_VEL
LIN {X 0,Y 428.299,Z 1150.651,A -85,B 0,C 180,E1 16102.906,E2 16102.906} C_VEL
LIN {X 0,Y 428.261,Z 1154.392,A -85,B 0,C 180,E1 16107.977,E2 16107.977} C_VEL
LIN {X 0,Y 428.216,Z 1154.434,A -85,B 0,C 180,E1 16112.021,E2 16112.021} C_VEL
LIN {X 0,Y 428.356,Z 1149.776,A -85,B 0,C 180,E1 16118.111,E2 16118.111} C_VEL
LIN {X 0,Y 429.299,Z 1140.497,A -85,B 0,C 180,E1 16123.743,E2 16123.743} C_VEL
LIN {X 0,Y 432.03,Z 1124.985,A -85,B 0,C 180,E1 16129.685,E2 16129.685} C_VEL
LIN {X 0,Y 434.967,Z 1112.329,A -85,B 0,C 180,E1 16133.326,E2 16133.326} C_VEL
LIN {X 0,Y 433.204,Z 1104.835,A -85,B 0,C 180,E1 16135.41,E2 16135.41} C_VEL
LIN {X 0,Y 431.91,Z 1096.677,A -85,B 0,C 180,E1 16137.461,E2 16137.461} C_VEL
LIN {X 0,Y 440.262,Z 1069.673,A -85,B 0,C 180,E1 16142.551,E2 16142.551} C_VEL
LIN {X 0,Y 451.087,Z 1035.562,A -85,B 0,C 180,E1 16147.329,E2 16147.329} C_VEL
LIN {X 0,Y 462.699,Z 997.198,A -85,B 0,C 180,E1 16151.268,E2 16151.268} C_VEL
LIN {X 0,Y 473.275,Z 957.757,A -85,B 0,C 180,E1 16154.218,E2 16154.218} C_VEL
LIN {X 0,Y 482.251,Z 917.369,A -85,B 0,C 180,E1 16156.399,E2 16156.399} C_VEL
LIN {X 0,Y 485.608,Z 897.988,A -85,B 0,C 180,E1 16157.219,E2 16157.219} C_VEL
LIN {X 0,Y 472.412,Z 865.515,A -85,B 0,C 180,E1 16160.834,E2 16160.834} C_VEL
LIN {X 0,Y 456.314,Z 835.977,A -85,B 0,C 180,E1 16164.812,E2 16164.812} C_VEL
LIN {X 0,Y 440.09,Z 811.609,A -85,B 0,C 180,E1 16168.933,E2 16168.933} C_VEL
LIN {X 0,Y 431.388,Z 799.676,A -85,B 0,C 180,E1 16171.427,E2 16171.427} C_VEL
LIN {X 0,Y 427.493,Z 794.258,A -85,B 0,C 180,E1 16172.652,E2 16172.652} C_VEL
LIN {X 0,Y 422.938,Z 787.76,A -85,B 0,C 180,E1 16174.195,E2 16174.195} C_VEL
LIN {X 0,Y 419.058,Z 783.013,A -85,B 0,C 180,E1 16175.579,E2 16175.579} C_VEL
LIN {X 0,Y 418.77,Z 780.81,A -85,B 0,C 180,E1 16175.916,E2 16175.916} C_VEL
LIN {X 0,Y 419.034,Z 780.81,A -85,B 0,C 180,E1 16181.068,E2 16181.068} C_VEL
LIN {X 0,Y 419.398,Z 780.81,A -85,B 0,C 180,E1 16187.521,E2 16187.521} C_VEL
LIN {X 0,Y 419.753,Z 780.81,A -85,B 0,C 180,E1 16193.804,E2 16193.804} C_VEL
LIN {X 0,Y 420.266,Z 780.81,A -85,B 0,C 180,E1 16200.003,E2 16200.003} C_VEL
LIN {X 0,Y 419.817,Z 780.81,A -85,B 0,C 180,E1 16206.201,E2 16206.201} C_VEL
LIN {X 0,Y 419.441,Z 780.81,A -85,B 0,C 180,E1 16212.485,E2 16212.485} C_VEL
LIN {X 0,Y 419.045,Z 780.81,A -85,B 0,C 180,E1 16218.938,E2 16218.938} C_VEL
LIN {X 0,Y 418.875,Z 781.487,A -85,B 0,C 180,E1 16221.759,E2 16221.759} C_VEL
LIN {X 0,Y 421.154,Z 786.402,A -85,B 0,C 180,E1 16222.677,E2 16222.677} C_VEL
LIN {X 0,Y 424.359,Z 789.594,A -85,B 0,C 180,E1 16223.754,E2 16223.754} C_VEL
LIN {X 0,Y 439.16,Z 810.143,A -85,B 0,C 180,E1 16228.305,E2 16228.305} C_VEL
LIN {X 0,Y 454.947,Z 835.041,A -85,B 0,C 180,E1 16232.623,E2 16232.623} C_VEL
LIN {X 0,Y 470.065,Z 864.887,A -85,B 0,C 180,E1 16236.847,E2 16236.847} C_VEL
LIN {X 0,Y 481.575,Z 896.165,A -85,B 0,C 180,E1 16240.613,E2 16240.613} C_VEL
LIN {X 0,Y 482.201,Z 901.818,A -85,B 0,C 180,E1 16241.126,E2 16241.126} C_VEL
LIN {X 0,Y 472.899,Z 942.71,A -85,B 0,C 180,E1 16243.543,E2 16243.543} C_VEL
LIN {X 0,Y 461.723,Z 983.103,A -85,B 0,C 180,E1 16246.897,E2 16246.897} C_VEL
LIN {X 0,Y 450.968,Z 1017.355,A -85,B 0,C 180,E1 16250.769,E2 16250.769} C_VEL
LIN {X 0,Y 441.434,Z 1046.136,A -85,B 0,C 180,E1 16255.065,E2 16255.065} C_VEL
LIN {X 0,Y 432.866,Z 1072.018,A -85,B 0,C 180,E1 16260.169,E2 16260.169} C_VEL
LIN {X 0,Y 426.35,Z 1093.409,A -85,B 0,C 180,E1 16265.948,E2 16265.948} C_VEL
LIN {X 0,Y 422.751,Z 1108.644,A -85,B 0,C 180,E1 16271.775,E2 16271.775} C_VEL
LIN {X 0,Y 420.846,Z 1118.661,A -85,B 0,C 180,E1 16277.56,E2 16277.56} C_VEL
LIN {X 0,Y 420.161,Z 1123.896,A -85,B 0,C 180,E1 16283.807,E2 16283.807} C_VEL
LIN {X 0,Y 420.396,Z 1123.731,A -85,B 0,C 180,E1 16290.001,E2 16290.001} C_VEL
LIN {X 0,Y 420.874,Z 1118.248,A -85,B 0,C 180,E1 16296.185,E2 16296.185} C_VEL
LIN {X 0,Y 422.724,Z 1107.054,A -85,B 0,C 180,E1 16302.386,E2 16302.386} C_VEL
LIN {X 0,Y 426.231,Z 1091.302,A -85,B 0,C 180,E1 16308.073,E2 16308.073} C_VEL
LIN {X 0,Y 432.013,Z 1070.752,A -85,B 0,C 180,E1 16313.447,E2 16313.447} C_VEL
LIN {X 0,Y 440.69,Z 1042.447,A -85,B 0,C 180,E1 16318.881,E2 16318.881} C_VEL
LIN {X 0,Y 450.963,Z 1009.267,A -85,B 0,C 180,E1 16323.566,E2 16323.566} C_VEL
LIN {X 0,Y 461.92,Z 970.96,A -85,B 0,C 180,E1 16327.54,E2 16327.54} C_VEL
LIN {X 0,Y 472.204,Z 928.553,A -85,B 0,C 180,E1 16330.736,E2 16330.736} C_VEL
LIN {X 0,Y 478.338,Z 897.292,A -85,B 0,C 180,E1 16332.493,E2 16332.493} C_VEL
LIN {X 0,Y 466.078,Z 862.678,A -85,B 0,C 180,E1 16336.253,E2 16336.253} C_VEL
LIN {X 0,Y 451.044,Z 831.879,A -85,B 0,C 180,E1 16340.045,E2 16340.045} C_VEL
LIN {X 0,Y 434.906,Z 805.894,A -85,B 0,C 180,E1 16343.876,E2 16343.876} C_VEL
LIN {X 0,Y 421.881,Z 787.289,A -85,B 0,C 180,E1 16347.184,E2 16347.184} C_VEL
LIN {X 0,Y 418.75,Z 782.671,A -85,B 0,C 180,E1 16348.061,E2 16348.061} C_VEL
LIN {X 0,Y 418.543,Z 780.81,A -85,B 0,C 180,E1 16348.291,E2 16348.291} C_VEL
LIN {X 0,Y 418.729,Z 780.81,A -85,B 0,C 180,E1 16354.451,E2 16354.451} C_VEL
LIN {X 0,Y 419.051,Z 780.81,A -85,B 0,C 180,E1 16361.062,E2 16361.062} C_VEL
LIN {X 0,Y 419.403,Z 780.81,A -85,B 0,C 180,E1 16367.514,E2 16367.514} C_VEL
LIN {X 0,Y 419.777,Z 780.81,A -85,B 0,C 180,E1 16373.798,E2 16373.798} C_VEL
LIN {X 0,Y 420.285,Z 780.81,A -85,B 0,C 180,E1 16379.997,E2 16379.997} C_VEL
LIN {X 0,Y 419.78,Z 780.81,A -85,B 0,C 180,E1 16386.195,E2 16386.195} C_VEL
LIN {X 0,Y 419.434,Z 780.81,A -85,B 0,C 180,E1 16392.478,E2 16392.478} C_VEL
LIN {X 0,Y 419.068,Z 780.81,A -85,B 0,C 180,E1 16398.93,E2 16398.93} C_VEL
LIN {X 0,Y 418.752,Z 780.81,A -85,B 0,C 180,E1 16405.652,E2 16405.652} C_VEL
LIN {X 0,Y 418.653,Z 781.251,A -85,B 0,C 180,E1 16408.329,E2 16408.329} C_VEL
LIN {X 0,Y 420.912,Z 786.388,A -85,B 0,C 180,E1 16409.026,E2 16409.026} C_VEL
LIN {X 0,Y 423.737,Z 789.712,A -85,B 0,C 180,E1 16409.77,E2 16409.77} C_VEL
LIN {X 0,Y 441.175,Z 814.872,A -85,B 0,C 180,E1 16413.998,E2 16413.998} C_VEL
LIN {X 0,Y 459.946,Z 846.553,A -85,B 0,C 180,E1 16418.09,E2 16418.09} C_VEL
LIN {X 0,Y 475.717,Z 880.721,A -85,B 0,C 180,E1 16421.752,E2 16421.752} C_VEL
LIN {X 0,Y 481.232,Z 897.808,A -85,B 0,C 180,E1 16423.336,E2 16423.336} C_VEL
LIN {X 0,Y 473.432,Z 939.832,A -85,B 0,C 180,E1 16425.27,E2 16425.27} C_VEL
LIN {X 0,Y 463.527,Z 982.215,A -85,B 0,C 180,E1 16428.064,E2 16428.064} C_VEL
LIN {X 0,Y 452.698,Z 1022.001,A -85,B 0,C 180,E1 16431.712,E2 16431.712} C_VEL
LIN {X 0,Y 442.07,Z 1058.282,A -85,B 0,C 180,E1 16436.256,E2 16436.256} C_VEL
LIN {X 0,Y 433.19,Z 1088.355,A -85,B 0,C 180,E1 16441.337,E2 16441.337} C_VEL
LIN {X 0,Y 427.022,Z 1111.441,A -85,B 0,C 180,E1 16446.54,E2 16446.54} C_VEL
LIN {X 0,Y 422.914,Z 1130.425,A -85,B 0,C 180,E1 16452.318,E2 16452.318} C_VEL
LIN {X 0,Y 420.813,Z 1144.492,A -85,B 0,C 180,E1 16458.608,E2 16458.608} C_VEL
LIN {X 0,Y 420.341,Z 1151.406,A -85,B 0,C 180,E1 16463.808,E2 16463.808} C_VEL
LIN {X 0,Y 420.36,Z 1154.107,A -85,B 0,C 180,E1 16467.939,E2 16467.939} C_VEL
LIN {X 0,Y 420.319,Z 1154.156,A -85,B 0,C 180,E1 16472.059,E2 16472.059} C_VEL
LIN {X 0,Y 420.478,Z 1149.516,A -85,B 0,C 180,E1 16478.264,E2 16478.264} C_VEL
LIN {X 0,Y 421.51,Z 1140.258,A -85,B 0,C 180,E1 16484.003,E2 16484.003} C_VEL
LIN {X 0,Y 424.429,Z 1124.532,A -85,B 0,C 180,E1 16490.132,E2 16490.132} C_VEL
LIN {X 0,Y 429.85,Z 1103.749,A -85,B 0,C 180,E1 16495.854,E2 16495.854} C_VEL
LIN {X 0,Y 431.91,Z 1096.677,A -85,B 0,C 180,E1 16497.461,E2 16497.461} C_VEL
LIN {X 0,Y 431.037,Z 1088.135,A -85,B 0,C 180,E1 16499.489,E2 16499.489} C_VEL
LIN {X 0,Y 430.349,Z 1078.991,A -85,B 0,C 180,E1 16501.479,E2 16501.479} C_VEL
LIN {X 0,Y 440.955,Z 1046.865,A -85,B 0,C 180,E1 16506.505,E2 16506.505} C_VEL
LIN {X 0,Y 452.892,Z 1009.878,A -85,B 0,C 180,E1 16510.745,E2 16510.745} C_VEL
LIN {X 0,Y 464.229,Z 970.528,A -85,B 0,C 180,E1 16514.045,E2 16514.045} C_VEL
LIN {X 0,Y 474.024,Z 930.277,A -85,B 0,C 180,E1 16516.486,E2 16516.486} C_VEL
LIN {X 0,Y 479.864,Z 901.681,A -85,B 0,C 180,E1 16517.756,E2 16517.756} C_VEL
LIN {X 0,Y 468.17,Z 871.412,A -85,B 0,C 180,E1 16521.214,E2 16521.214} C_VEL
LIN {X 0,Y 452.966,Z 842.567,A -85,B 0,C 180,E1 16525.17,E2 16525.17} C_VEL
LIN {X 0,Y 435.383,Z 815.086,A -85,B 0,C 180,E1 16529.911,E2 16529.911} C_VEL
LIN {X 0,Y 424.344,Z 800.438,A -85,B 0,C 180,E1 16533.292,E2 16533.292} C_VEL
LIN {X 0,Y 420.283,Z 794.711,A -85,B 0,C 180,E1 16534.71,E2 16534.71} C_VEL
LIN {X 0,Y 416.331,Z 788.794,A -85,B 0,C 180,E1 16536.214,E2 16536.214} C_VEL
LIN {X 0,Y 411.403,Z 783.508,A -85,B 0,C 180,E1 16538.179,E2 16538.179} C_VEL
LIN {X 0,Y 411.009,Z 780.81,A -85,B 0,C 180,E1 16538.645,E2 16538.645} C_VEL
LIN {X 0,Y 411.331,Z 780.81,A -85,B 0,C 180,E1 16545.104,E2 16545.104} C_VEL
LIN {X 0,Y 411.76,Z 780.81,A -85,B 0,C 180,E1 16552.24,E2 16552.24} C_VEL
LIN {X 0,Y 412.183,Z 780.81,A -85,B 0,C 180,E1 16557.903,E2 16557.903} C_VEL
LIN {X 0,Y 412.204,Z 780.81,A -85,B 0,C 180,E1 16562.104,E2 16562.104} C_VEL
LIN {X 0,Y 411.812,Z 780.81,A -85,B 0,C 180,E1 16568.442,E2 16568.442} C_VEL
LIN {X 0,Y 411.38,Z 780.81,A -85,B 0,C 180,E1 16574.9,E2 16574.9} C_VEL
LIN {X 0,Y 411.143,Z 780.81,A -85,B 0,C 180,E1 16579.037,E2 16579.037} C_VEL
LIN {X 0,Y 412.884,Z 785.859,A -85,B 0,C 180,E1 16579.932,E2 16579.932} C_VEL
LIN {X 0,Y 416.552,Z 789.211,A -85,B 0,C 180,E1 16581.339,E2 16581.339} C_VEL
LIN {X 0,Y 420.609,Z 794.875,A -85,B 0,C 180,E1 16582.858,E2 16582.858} C_VEL
LIN {X 0,Y 435.667,Z 815.695,A -85,B 0,C 180,E1 16587.708,E2 16587.708} C_VEL
LIN {X 0,Y 452.492,Z 843.525,A -85,B 0,C 180,E1 16592.611,E2 16592.611} C_VEL
LIN {X 0,Y 466.506,Z 873.058,A -85,B 0,C 180,E1 16596.813,E2 16596.813} C_VEL
LIN {X 0,Y 476.623,Z 902.838,A -85,B 0,C 180,E1 16600.458,E2 16600.458} C_VEL
LIN {X 0,Y 466.915,Z 944.273,A -85,B 0,C 180,E1 16602.948,E2 16602.948} C_VEL
LIN {X 0,Y 455.368,Z 984.557,A -85,B 0,C 180,E1 16606.34,E2 16606.34} C_VEL
LIN {X 0,Y 443.456,Z 1021.217,A -85,B 0,C 180,E1 16610.607,E2 16610.607} C_VEL
LIN {X 0,Y 432.796,Z 1051.744,A -85,B 0,C 180,E1 16615.425,E2 16615.425} C_VEL
LIN {X 0,Y 424.263,Z 1076.536,A -85,B 0,C 180,E1 16620.695,E2 16620.695} C_VEL
LIN {X 0,Y 418.032,Z 1096.785,A -85,B 0,C 180,E1 16626.571,E2 16626.571} C_VEL
LIN {X 0,Y 414.733,Z 1110.211,A -85,B 0,C 180,E1 16632.073,E2 16632.073} C_VEL
LIN {X 0,Y 413.028,Z 1118.896,A -85,B 0,C 180,E1 16637.321,E2 16637.321} C_VEL
LIN {X 0,Y 412.262,Z 1124.161,A -85,B 0,C 180,E1 16643.688,E2 16643.688} C_VEL
LIN {X 0,Y 412.499,Z 1124.029,A -85,B 0,C 180,E1 16650.001,E2 16650.001} C_VEL
LIN {X 0,Y 413.004,Z 1118.583,A -85,B 0,C 180,E1 16656.303,E2 16656.303} C_VEL
LIN {X 0,Y 414.954,Z 1107.414,A -85,B 0,C 180,E1 16662.622,E2 16662.622} C_VEL
LIN {X 0,Y 418.621,Z 1091.704,A -85,B 0,C 180,E1 16668.413,E2 16668.413} C_VEL
LIN {X 0,Y 424.691,Z 1071.196,A -85,B 0,C 180,E1 16673.876,E2 16673.876} C_VEL
LIN {X 0,Y 433.385,Z 1043.971,A -85,B 0,C 180,E1 16679.22,E2 16679.22} C_VEL
LIN {X 0,Y 444.355,Z 1009.803,A -85,B 0,C 180,E1 16684.134,E2 16684.134} C_VEL
LIN {X 0,Y 455.669,Z 971.568,A -85,B 0,C 180,E1 16688.146,E2 16688.146} C_VEL
LIN {X 0,Y 466.351,Z 928.944,A -85,B 0,C 180,E1 16691.387,E2 16691.387} C_VEL
LIN {X 0,Y 472.028,Z 899.773,A -85,B 0,C 180,E1 16693.079,E2 16693.079} C_VEL
LIN {X 0,Y 460.395,Z 866.144,A -85,B 0,C 180,E1 16696.87,E2 16696.87} C_VEL
LIN {X 0,Y 445.761,Z 835.375,A -85,B 0,C 180,E1 16700.783,E2 16700.783} C_VEL
LIN {X 0,Y 427.921,Z 806.718,A -85,B 0,C 180,E1 16705.25,E2 16705.25} C_VEL
LIN {X 0,Y 417.88,Z 792.936,A -85,B 0,C 180,E1 16707.922,E2 16707.922} C_VEL
LIN {X 0,Y 414.247,Z 787.462,A -85,B 0,C 180,E1 16708.988,E2 16708.988} C_VEL
LIN {X 0,Y 410.938,Z 782.724,A -85,B 0,C 180,E1 16709.998,E2 16709.998} C_VEL
LIN {X 0,Y 410.69,Z 780.81,A -85,B 0,C 180,E1 16710.221,E2 16710.221} C_VEL
LIN {X 0,Y 410.936,Z 780.81,A -85,B 0,C 180,E1 16716.828,E2 16716.828} C_VEL
LIN {X 0,Y 411.221,Z 780.81,A -85,B 0,C 180,E1 16722.904,E2 16722.904} C_VEL
LIN {X 0,Y 411.589,Z 780.81,A -85,B 0,C 180,E1 16729.421,E2 16729.421} C_VEL
LIN {X 0,Y 412.059,Z 780.81,A -85,B 0,C 180,E1 16735.791,E2 16735.791} C_VEL
LIN {X 0,Y 412.216,Z 780.81,A -85,B 0,C 180,E1 16742.097,E2 16742.097} C_VEL
LIN {X 0,Y 411.769,Z 780.81,A -85,B 0,C 180,E1 16748.436,E2 16748.436} C_VEL
LIN {X 0,Y 411.368,Z 780.81,A -85,B 0,C 180,E1 16754.894,E2 16754.894} C_VEL
LIN {X 0,Y 410.979,Z 780.81,A -85,B 0,C 180,E1 16761.566,E2 16761.566} C_VEL
LIN {X 0,Y 410.764,Z 780.877,A -85,B 0,C 180,E1 16766.349,E2 16766.349} C_VEL
LIN {X 0,Y 412.659,Z 785.998,A -85,B 0,C 180,E1 16767.022,E2 16767.022} C_VEL
LIN {X 0,Y 415.874,Z 789.45,A -85,B 0,C 180,E1 16767.94,E2 16767.94} C_VEL
LIN {X 0,Y 433.617,Z 814.82,A -85,B 0,C 180,E1 16772.578,E2 16772.578} C_VEL
LIN {X 0,Y 452.029,Z 845.213,A -85,B 0,C 180,E1 16776.818,E2 16776.818} C_VEL
LIN {X 0,Y 468.217,Z 879.694,A -85,B 0,C 180,E1 16780.727,E2 16780.727} C_VEL
LIN {X 0,Y 475.26,Z 899.976,A -85,B 0,C 180,E1 16782.745,E2 16782.745} C_VEL
LIN {X 0,Y 467.39,Z 940.677,A -85,B 0,C 180,E1 16784.66,E2 16784.66} C_VEL
LIN {X 0,Y 457.535,Z 981.647,A -85,B 0,C 180,E1 16787.385,E2 16787.385} C_VEL
LIN {X 0,Y 445.996,Z 1022.581,A -85,B 0,C 180,E1 16791.177,E2 16791.177} C_VEL
LIN {X 0,Y 435.284,Z 1057.829,A -85,B 0,C 180,E1 16795.657,E2 16795.657} C_VEL
LIN {X 0,Y 425.991,Z 1087.942,A -85,B 0,C 180,E1 16800.806,E2 16800.806} C_VEL
LIN {X 0,Y 419.498,Z 1111.058,A -85,B 0,C 180,E1 16806.092,E2 16806.092} C_VEL
LIN {X 0,Y 415.171,Z 1130.078,A -85,B 0,C 180,E1 16811.977,E2 16811.977} C_VEL
LIN {X 0,Y 413.175,Z 1142.19,A -85,B 0,C 180,E1 16817.323,E2 16817.323} C_VEL
LIN {X 0,Y 412.514,Z 1150.036,A -85,B 0,C 180,E1 16822.633,E2 16822.633} C_VEL
LIN {X 0,Y 412.456,Z 1153.82,A -85,B 0,C 180,E1 16827.899,E2 16827.899} C_VEL
LIN {X 0,Y 412.415,Z 1153.878,A -85,B 0,C 180,E1 16832.099,E2 16832.099} C_VEL
LIN {X 0,Y 412.585,Z 1149.257,A -85,B 0,C 180,E1 16838.423,E2 16838.423} C_VEL
LIN {X 0,Y 413.688,Z 1140.017,A -85,B 0,C 180,E1 16844.273,E2 16844.273} C_VEL
LIN {X 0,Y 416.953,Z 1123.801,A -85,B 0,C 180,E1 16850.691,E2 16850.691} C_VEL
LIN {X 0,Y 422.677,Z 1103.05,A -85,B 0,C 180,E1 16856.458,E2 16856.458} C_VEL
LIN {X 0,Y 430.349,Z 1078.991,A -85,B 0,C 180,E1 16861.479,E2 16861.479} C_VEL
LIN {X 0,Y 429.995,Z 1069.465,A -85,B 0,C 180,E1 16863.426,E2 16863.426} C_VEL
LIN {X 0,Y 430.152,Z 1059.241,A -85,B 0,C 180,E1 16865.34,E2 16865.34} C_VEL
LIN {X 0,Y 441.684,Z 1025.253,A -85,B 0,C 180,E1 16869.79,E2 16869.79} C_VEL
LIN {X 0,Y 453.273,Z 988.64,A -85,B 0,C 180,E1 16873.339,E2 16873.339} C_VEL
LIN {X 0,Y 463.96,Z 949.999,A -85,B 0,C 180,E1 16876.103,E2 16876.103} C_VEL
LIN {X 0,Y 473.968,Z 905.421,A -85,B 0,C 180,E1 16878.327,E2 16878.327} C_VEL
LIN {X 0,Y 465.001,Z 880.277,A -85,B 0,C 180,E1 16881.207,E2 16881.207} C_VEL
LIN {X 0,Y 450.202,Z 850.085,A -85,B 0,C 180,E1 16885.364,E2 16885.364} C_VEL
LIN {X 0,Y 432.709,Z 821.929,A -85,B 0,C 180,E1 16890.309,E2 16890.309} C_VEL
LIN {X 0,Y 421.439,Z 806.706,A -85,B 0,C 180,E1 16893.882,E2 16893.882} C_VEL
LIN {X 0,Y 417.335,Z 801.17,A -85,B 0,C 180,E1 16895.355,E2 16895.355} C_VEL
LIN {X 0,Y 413.003,Z 795.102,A -85,B 0,C 180,E1 16897.058,E2 16897.058} C_VEL
LIN {X 0,Y 408.979,Z 789.614,A -85,B 0,C 180,E1 16898.791,E2 16898.791} C_VEL
LIN {X 0,Y 407.439,Z 787.846,A -85,B 0,C 180,E1 16899.487,E2 16899.487} C_VEL
LIN {X 0,Y 403.48,Z 782.969,A -85,B 0,C 180,E1 16901.444,E2 16901.444} C_VEL
LIN {X 0,Y 403.213,Z 780.81,A -85,B 0,C 180,E1 16901.714,E2 16901.714} C_VEL
LIN {X 0,Y 403.538,Z 780.81,A -85,B 0,C 180,E1 16907.022,E2 16907.022} C_VEL
LIN {X 0,Y 403.942,Z 780.81,A -85,B 0,C 180,E1 16913.561,E2 16913.561} C_VEL
LIN {X 0,Y 404.461,Z 780.81,A -85,B 0,C 180,E1 16920.003,E2 16920.003} C_VEL
LIN {X 0,Y 404.002,Z 780.81,A -85,B 0,C 180,E1 16926.445,E2 16926.445} C_VEL
LIN {X 0,Y 403.56,Z 780.81,A -85,B 0,C 180,E1 16933.212,E2 16933.212} C_VEL
LIN {X 0,Y 403.395,Z 781.441,A -85,B 0,C 180,E1 16935.889,E2 16935.889} C_VEL
LIN {X 0,Y 405.451,Z 786.168,A -85,B 0,C 180,E1 16937.064,E2 16937.064} C_VEL
LIN {X 0,Y 409.121,Z 789.438,A -85,B 0,C 180,E1 16938.716,E2 16938.716} C_VEL
LIN {X 0,Y 413.028,Z 795.014,A -85,B 0,C 180,E1 16940.408,E2 16940.408} C_VEL
LIN {X 0,Y 420.926,Z 805.917,A -85,B 0,C 180,E1 16943.399,E2 16943.399} C_VEL
LIN {X 0,Y 433.02,Z 822.884,A -85,B 0,C 180,E1 16947.384,E2 16947.384} C_VEL
LIN {X 0,Y 448.639,Z 849.641,A -85,B 0,C 180,E1 16952.21,E2 16952.21} C_VEL
LIN {X 0,Y 461.64,Z 878.251,A -85,B 0,C 180,E1 16956.387,E2 16956.387} C_VEL
LIN {X 0,Y 470.557,Z 905.233,A -85,B 0,C 180,E1 16959.807,E2 16959.807} C_VEL
LIN {X 0,Y 460.903,Z 946.064,A -85,B 0,C 180,E1 16962.354,E2 16962.354} C_VEL
LIN {X 0,Y 449.161,Z 985.634,A -85,B 0,C 180,E1 16965.737,E2 16965.737} C_VEL
LIN {X 0,Y 437.017,Z 1021.572,A -85,B 0,C 180,E1 16969.964,E2 16969.964} C_VEL
LIN {X 0,Y 425.755,Z 1052.664,A -85,B 0,C 180,E1 16974.946,E2 16974.946} C_VEL
LIN {X 0,Y 416.63,Z 1078.113,A -85,B 0,C 180,E1 16980.503,E2 16980.503} C_VEL
LIN {X 0,Y 410.501,Z 1096.972,A -85,B 0,C 180,E1 16986.115,E2 16986.115} C_VEL
LIN {X 0,Y 406.989,Z 1110.602,A -85,B 0,C 180,E1 16991.81,E2 16991.81} C_VEL
LIN {X 0,Y 405.19,Z 1119.131,A -85,B 0,C 180,E1 16997.071,E2 16997.071} C_VEL
LIN {X 0,Y 404.364,Z 1124.427,A -85,B 0,C 180,E1 17003.564,E2 17003.564} C_VEL
LIN {X 0,Y 404.615,Z 1124.327,A -85,B 0,C 180,E1 17010.001,E2 17010.001} C_VEL
LIN {X 0,Y 405.148,Z 1118.916,A -85,B 0,C 180,E1 17016.426,E2 17016.426} C_VEL
LIN {X 0,Y 407.202,Z 1107.773,A -85,B 0,C 180,E1 17022.866,E2 17022.866} C_VEL
LIN {X 0,Y 411.039,Z 1092.104,A -85,B 0,C 180,E1 17028.766,E2 17028.766} C_VEL
LIN {X 0,Y 417.377,Z 1071.64,A -85,B 0,C 180,E1 17034.321,E2 17034.321} C_VEL
LIN {X 0,Y 426.42,Z 1044.446,A -85,B 0,C 180,E1 17039.745,E2 17039.745} C_VEL
LIN {X 0,Y 437.171,Z 1012.214,A -85,B 0,C 180,E1 17044.474,E2 17044.474} C_VEL
LIN {X 0,Y 447.982,Z 977.125,A -85,B 0,C 180,E1 17048.304,E2 17048.304} C_VEL
LIN {X 0,Y 458.156,Z 939.148,A -85,B 0,C 180,E1 17051.396,E2 17051.396} C_VEL
LIN {X 0,Y 466.039,Z 903.229,A -85,B 0,C 180,E1 17053.567,E2 17053.567} C_VEL
LIN {X 0,Y 455.717,Z 872.05,A -85,B 0,C 180,E1 17057.179,E2 17057.179} C_VEL
LIN {X 0,Y 441.594,Z 841.244,A -85,B 0,C 180,E1 17061.201,E2 17061.201} C_VEL
LIN {X 0,Y 424.696,Z 813.159,A -85,B 0,C 180,E1 17065.693,E2 17065.693} C_VEL
LIN {X 0,Y 411.1,Z 794.003,A -85,B 0,C 180,E1 17069.55,E2 17069.55} C_VEL
LIN {X 0,Y 406.5,Z 787.528,A -85,B 0,C 180,E1 17071.009,E2 17071.009} C_VEL
LIN {X 0,Y 403.056,Z 782.686,A -85,B 0,C 180,E1 17072.173,E2 17072.173} C_VEL
LIN {X 0,Y 402.812,Z 780.81,A -85,B 0,C 180,E1 17072.374,E2 17072.374} C_VEL
LIN {X 0,Y 403.105,Z 780.81,A -85,B 0,C 180,E1 17079.584,E2 17079.584} C_VEL
LIN {X 0,Y 403.531,Z 780.81,A -85,B 0,C 180,E1 17086.816,E2 17086.816} C_VEL
LIN {X 0,Y 403.966,Z 780.81,A -85,B 0,C 180,E1 17093.554,E2 17093.554} C_VEL
LIN {X 0,Y 404.48,Z 780.81,A -85,B 0,C 180,E1 17099.997,E2 17099.997} C_VEL
LIN {X 0,Y 403.967,Z 780.81,A -85,B 0,C 180,E1 17106.439,E2 17106.439} C_VEL
LIN {X 0,Y 403.539,Z 780.81,A -85,B 0,C 180,E1 17113.189,E2 17113.189} C_VEL
LIN {X 0,Y 403.165,Z 780.81,A -85,B 0,C 180,E1 17119.707,E2 17119.707} C_VEL
LIN {X 0,Y 402.954,Z 781.341,A -85,B 0,C 180,E1 17124.203,E2 17124.203} C_VEL
LIN {X 0,Y 405.195,Z 786.441,A -85,B 0,C 180,E1 17125.047,E2 17125.047} C_VEL
LIN {X 0,Y 408.188,Z 789.512,A -85,B 0,C 180,E1 17125.984,E2 17125.984} C_VEL
LIN {X 0,Y 423.529,Z 811.266,A -85,B 0,C 180,E1 17130.405,E2 17130.405} C_VEL
LIN {X 0,Y 440.565,Z 837.676,A -85,B 0,C 180,E1 17134.594,E2 17134.594} C_VEL
LIN {X 0,Y 457.298,Z 870.509,A -85,B 0,C 180,E1 17138.727,E2 17138.727} C_VEL
LIN {X 0,Y 469.284,Z 902.102,A -85,B 0,C 180,E1 17142.13,E2 17142.13} C_VEL
LIN {X 0,Y 460.836,Z 943.985,A -85,B 0,C 180,E1 17144.177,E2 17144.177} C_VEL
LIN {X 0,Y 450.787,Z 983.918,A -85,B 0,C 180,E1 17146.92,E2 17146.92} C_VEL
LIN {X 0,Y 439.688,Z 1022.087,A -85,B 0,C 180,E1 17150.513,E2 17150.513} C_VEL
LIN {X 0,Y 428.487,Z 1057.473,A -85,B 0,C 180,E1 17155.051,E2 17155.051} C_VEL
LIN {X 0,Y 418.87,Z 1087.623,A -85,B 0,C 180,E1 17160.281,E2 17160.281} C_VEL
LIN {X 0,Y 411.996,Z 1110.677,A -85,B 0,C 180,E1 17165.629,E2 17165.629} C_VEL
LIN {X 0,Y 407.43,Z 1129.871,A -85,B 0,C 180,E1 17171.68,E2 17171.68} C_VEL
LIN {X 0,Y 405.111,Z 1143.84,A -85,B 0,C 180,E1 17178.16,E2 17178.16} C_VEL
LIN {X 0,Y 404.547,Z 1150.805,A -85,B 0,C 180,E1 17183.565,E2 17183.565} C_VEL
LIN {X 0,Y 404.551,Z 1153.532,A -85,B 0,C 180,E1 17187.858,E2 17187.858} C_VEL
LIN {X 0,Y 404.511,Z 1153.6,A -85,B 0,C 180,E1 17192.14,E2 17192.14} C_VEL
LIN {X 0,Y 404.716,Z 1149,A -85,B 0,C 180,E1 17198.588,E2 17198.588} C_VEL
LIN {X 0,Y 405.906,Z 1139.679,A -85,B 0,C 180,E1 17204.601,E2 17204.601} C_VEL
LIN {X 0,Y 409.377,Z 1123.578,A -85,B 0,C 180,E1 17211.092,E2 17211.092} C_VEL
LIN {X 0,Y 415.564,Z 1102.157,A -85,B 0,C 180,E1 17217.133,E2 17217.133} C_VEL
LIN {X 0,Y 423.868,Z 1077.331,A -85,B 0,C 180,E1 17222.326,E2 17222.326} C_VEL
LIN {X 0,Y 430.152,Z 1059.241,A -85,B 0,C 180,E1 17225.34,E2 17225.34} C_VEL
LIN {X 0,Y 430.491,Z 1048.665,A -85,B 0,C 180,E1 17227.204,E2 17227.204} C_VEL
LIN {X 0,Y 431.146,Z 1037.5,A -85,B 0,C 180,E1 17228.997,E2 17228.997} C_VEL
LIN {X 0,Y 443.207,Z 1001.975,A -85,B 0,C 180,E1 17232.866,E2 17232.866} C_VEL
LIN {X 0,Y 454.843,Z 963.638,A -85,B 0,C 180,E1 17235.939,E2 17235.939} C_VEL
LIN {X 0,Y 465.281,Z 922.007,A -85,B 0,C 180,E1 17238.328,E2 17238.328} C_VEL
LIN {X 0,Y 468.092,Z 907.046,A -85,B 0,C 180,E1 17239.037,E2 17239.037} C_VEL
LIN {X 0,Y 456.635,Z 876.997,A -85,B 0,C 180,E1 17242.768,E2 17242.768} C_VEL
LIN {X 0,Y 442.415,Z 849.108,A -85,B 0,C 180,E1 17246.956,E2 17246.956} C_VEL
LIN {X 0,Y 427.775,Z 825.789,A -85,B 0,C 180,E1 17251.383,E2 17251.383} C_VEL
LIN {X 0,Y 415.625,Z 808.731,A -85,B 0,C 180,E1 17255.578,E2 17255.578} C_VEL
LIN {X 0,Y 410.411,Z 801.948,A -85,B 0,C 180,E1 17257.656,E2 17257.656} C_VEL
LIN {X 0,Y 405.7,Z 795.351,A -85,B 0,C 180,E1 17259.797,E2 17259.797} C_VEL
LIN {X 0,Y 401.561,Z 789.887,A -85,B 0,C 180,E1 17261.92,E2 17261.92} C_VEL
LIN {X 0,Y 399.996,Z 787.992,A -85,B 0,C 180,E1 17262.797,E2 17262.797} C_VEL
LIN {X 0,Y 395.916,Z 783.346,A -85,B 0,C 180,E1 17265.359,E2 17265.359} C_VEL
LIN {X 0,Y 395.507,Z 780.81,A -85,B 0,C 180,E1 17265.909,E2 17265.909} C_VEL
LIN {X 0,Y 395.939,Z 780.81,A -85,B 0,C 180,E1 17272.871,E2 17272.871} C_VEL
LIN {X 0,Y 396.558,Z 780.81,A -85,B 0,C 180,E1 17280.003,E2 17280.003} C_VEL
LIN {X 0,Y 396.005,Z 780.81,A -85,B 0,C 180,E1 17287.205,E2 17287.205} C_VEL
LIN {X 0,Y 395.718,Z 781.593,A -85,B 0,C 180,E1 17291.846,E2 17291.846} C_VEL
LIN {X 0,Y 398.188,Z 786.665,A -85,B 0,C 180,E1 17293.64,E2 17293.64} C_VEL
LIN {X 0,Y 401.526,Z 789.224,A -85,B 0,C 180,E1 17295.485,E2 17295.485} C_VEL
LIN {X 0,Y 405.049,Z 794.786,A -85,B 0,C 180,E1 17297.365,E2 17297.365} C_VEL
LIN {X 0,Y 407.262,Z 797.119,A -85,B 0,C 180,E1 17298.384,E2 17298.384} C_VEL
LIN {X 0,Y 413.233,Z 805.568,A -85,B 0,C 180,E1 17300.957,E2 17300.957} C_VEL
LIN {X 0,Y 422.347,Z 818.065,A -85,B 0,C 180,E1 17304.374,E2 17304.374} C_VEL
LIN {X 0,Y 436.78,Z 840.981,A -85,B 0,C 180,E1 17309.236,E2 17309.236} C_VEL
LIN {X 0,Y 450.718,Z 868.524,A -85,B 0,C 180,E1 17313.807,E2 17313.807} C_VEL
LIN {X 0,Y 461.933,Z 898.514,A -85,B 0,C 180,E1 17317.964,E2 17317.964} C_VEL
LIN {X 0,Y 464.549,Z 910.563,A -85,B 0,C 180,E1 17319.388,E2 17319.388} C_VEL
LIN {X 0,Y 454.609,Z 948.995,A -85,B 0,C 180,E1 17321.83,E2 17321.83} C_VEL
LIN {X 0,Y 443.035,Z 986.565,A -85,B 0,C 180,E1 17325.1,E2 17325.1} C_VEL
LIN {X 0,Y 430.442,Z 1022.53,A -85,B 0,C 180,E1 17329.387,E2 17329.387} C_VEL
LIN {X 0,Y 418.666,Z 1053.822,A -85,B 0,C 180,E1 17334.495,E2 17334.495} C_VEL
LIN {X 0,Y 408.856,Z 1080.028,A -85,B 0,C 180,E1 17340.387,E2 17340.387} C_VEL
LIN {X 0,Y 402.573,Z 1098.688,A -85,B 0,C 180,E1 17346.211,E2 17346.211} C_VEL
LIN {X 0,Y 398.863,Z 1112.571,A -85,B 0,C 180,E1 17352.358,E2 17352.358} C_VEL
LIN {X 0,Y 396.963,Z 1121.753,A -85,B 0,C 180,E1 17359.029,E2 17359.029} C_VEL
LIN {X 0,Y 396.468,Z 1124.692,A -85,B 0,C 180,E1 17363.436,E2 17363.436} C_VEL
LIN {X 0,Y 396.717,Z 1124.625,A -85,B 0,C 180,E1 17370.001,E2 17370.001} C_VEL
LIN {X 0,Y 397.28,Z 1119.25,A -85,B 0,C 180,E1 17376.553,E2 17376.553} C_VEL
LIN {X 0,Y 399.454,Z 1108.132,A -85,B 0,C 180,E1 17383.12,E2 17383.12} C_VEL
LIN {X 0,Y 403.48,Z 1092.503,A -85,B 0,C 180,E1 17389.131,E2 17389.131} C_VEL
LIN {X 0,Y 410.407,Z 1071.085,A -85,B 0,C 180,E1 17395.01,E2 17395.01} C_VEL
LIN {X 0,Y 420.06,Z 1043.424,A -85,B 0,C 180,E1 17400.54,E2 17400.54} C_VEL
LIN {X 0,Y 431.276,Z 1010.867,A -85,B 0,C 180,E1 17405.32,E2 17405.32} C_VEL
LIN {X 0,Y 442.951,Z 974.01,A -85,B 0,C 180,E1 17409.292,E2 17409.292} C_VEL
LIN {X 0,Y 453.566,Z 934.577,A -85,B 0,C 180,E1 17412.418,E2 17412.418} C_VEL
LIN {X 0,Y 459.922,Z 906.129,A -85,B 0,C 180,E1 17414.134,E2 17414.134} C_VEL
LIN {X 0,Y 449.459,Z 873.982,A -85,B 0,C 180,E1 17417.994,E2 17417.994} C_VEL
LIN {X 0,Y 435.175,Z 842.806,A -85,B 0,C 180,E1 17422.269,E2 17422.269} C_VEL
LIN {X 0,Y 417.907,Z 814.096,A -85,B 0,C 180,E1 17427.157,E2 17427.157} C_VEL
LIN {X 0,Y 403.985,Z 794.544,A -85,B 0,C 180,E1 17431.44,E2 17431.44} C_VEL
LIN {X 0,Y 398.935,Z 787.673,A -85,B 0,C 180,E1 17433.207,E2 17433.207} C_VEL
LIN {X 0,Y 395.261,Z 783.014,A -85,B 0,C 180,E1 17434.584,E2 17434.584} C_VEL
LIN {X 0,Y 394.933,Z 780.81,A -85,B 0,C 180,E1 17434.928,E2 17434.928} C_VEL
LIN {X 0,Y 395.332,Z 780.81,A -85,B 0,C 180,E1 17442.194,E2 17442.194} C_VEL
LIN {X 0,Y 395.722,Z 780.81,A -85,B 0,C 180,E1 17448.991,E2 17448.991} C_VEL
LIN {X 0,Y 396.227,Z 780.81,A -85,B 0,C 180,E1 17455.623,E2 17455.623} C_VEL
LIN {X 0,Y 396.577,Z 780.81,A -85,B 0,C 180,E1 17459.997,E2 17459.997} C_VEL
LIN {X 0,Y 395.962,Z 780.81,A -85,B 0,C 180,E1 17467.135,E2 17467.135} C_VEL
LIN {X 0,Y 395.645,Z 780.81,A -85,B 0,C 180,E1 17473.242,E2 17473.242} C_VEL
LIN {X 0,Y 395.223,Z 780.81,A -85,B 0,C 180,E1 17480.12,E2 17480.12} C_VEL
LIN {X 0,Y 395.137,Z 781.28,A -85,B 0,C 180,E1 17481.757,E2 17481.757} C_VEL
LIN {X 0,Y 397.434,Z 786.435,A -85,B 0,C 180,E1 17482.731,E2 17482.731} C_VEL
LIN {X 0,Y 400.425,Z 789.351,A -85,B 0,C 180,E1 17483.776,E2 17483.776} C_VEL
LIN {X 0,Y 404.724,Z 795.042,A -85,B 0,C 180,E1 17485.246,E2 17485.246} C_VEL
LIN {X 0,Y 423.254,Z 821.604,A -85,B 0,C 180,E1 17490.676,E2 17490.676} C_VEL
LIN {X 0,Y 440.294,Z 850.273,A -85,B 0,C 180,E1 17495.073,E2 17495.073} C_VEL
LIN {X 0,Y 455.077,Z 882.04,A -85,B 0,C 180,E1 17499.029,E2 17499.029} C_VEL
LIN {X 0,Y 463.293,Z 905.564,A -85,B 0,C 180,E1 17501.576,E2 17501.576} C_VEL
LIN {X 0,Y 454.003,Z 948.869,A -85,B 0,C 180,E1 17503.779,E2 17503.779} C_VEL
LIN {X 0,Y 443.248,Z 989.003,A -85,B 0,C 180,E1 17506.677,E2 17506.677} C_VEL
LIN {X 0,Y 432.094,Z 1025.542,A -85,B 0,C 180,E1 17510.281,E2 17510.281} C_VEL
LIN {X 0,Y 421.18,Z 1058.84,A -85,B 0,C 180,E1 17514.687,E2 17514.687} C_VEL
LIN {X 0,Y 411.175,Z 1089.029,A -85,B 0,C 180,E1 17520.076,E2 17520.076} C_VEL
LIN {X 0,Y 403.666,Z 1113.67,A -85,B 0,C 180,E1 17526.087,E2 17526.087} C_VEL
LIN {X 0,Y 399.17,Z 1132.127,A -85,B 0,C 180,E1 17532.37,E2 17532.37} C_VEL
LIN {X 0,Y 397.275,Z 1143.513,A -85,B 0,C 180,E1 17537.923,E2 17537.923} C_VEL
LIN {X 0,Y 396.655,Z 1150.504,A -85,B 0,C 180,E1 17543.436,E2 17543.436} C_VEL
LIN {X 0,Y 396.647,Z 1153.243,A -85,B 0,C 180,E1 17547.815,E2 17547.815} C_VEL
LIN {X 0,Y 396.607,Z 1153.322,A -85,B 0,C 180,E1 17552.182,E2 17552.182} C_VEL
LIN {X 0,Y 396.83,Z 1148.741,A -85,B 0,C 180,E1 17558.76,E2 17558.76} C_VEL
LIN {X 0,Y 398.033,Z 1139.794,A -85,B 0,C 180,E1 17564.701,E2 17564.701} C_VEL
LIN {X 0,Y 401.332,Z 1124.916,A -85,B 0,C 180,E1 17570.957,E2 17570.957} C_VEL
LIN {X 0,Y 407.275,Z 1105.215,A -85,B 0,C 180,E1 17576.847,E2 17576.847} C_VEL
LIN {X 0,Y 416.473,Z 1078.644,A -85,B 0,C 180,E1 17582.663,E2 17582.663} C_VEL
LIN {X 0,Y 428.199,Z 1045.927,A -85,B 0,C 180,E1 17587.9,E2 17587.9} C_VEL
LIN {X 0,Y 431.146,Z 1037.5,A -85,B 0,C 180,E1 17588.997,E2 17588.997} C_VEL
LIN {X 0,Y 432.201,Z 1025.892,A -85,B 0,C 180,E1 17590.739,E2 17590.739} C_VEL
LIN {X 0,Y 433.374,Z 1013.752,A -85,B 0,C 180,E1 17592.406,E2 17592.406} C_VEL
LIN {X 0,Y 445.582,Z 976.33,A -85,B 0,C 180,E1 17595.752,E2 17595.752} C_VEL
LIN {X 0,Y 457.114,Z 934.237,A -85,B 0,C 180,E1 17598.466,E2 17598.466} C_VEL
LIN {X 0,Y 462.188,Z 909.682,A -85,B 0,C 180,E1 17599.705,E2 17599.705} C_VEL
LIN {X 0,Y 450.641,Z 879.009,A -85,B 0,C 180,E1 17603.685,E2 17603.685} C_VEL
LIN {X 0,Y 436.441,Z 850.984,A -85,B 0,C 180,E1 17608.139,E2 17608.139} C_VEL
LIN {X 0,Y 422.143,Z 828.177,A -85,B 0,C 180,E1 17612.782,E2 17612.782} C_VEL
LIN {X 0,Y 412.717,Z 814.968,A -85,B 0,C 180,E1 17616.258,E2 17616.258} C_VEL
LIN {X 0,Y 408.045,Z 808.76,A -85,B 0,C 180,E1 17618.195,E2 17618.195} C_VEL
LIN {X 0,Y 403.711,Z 802.638,A -85,B 0,C 180,E1 17620.231,E2 17620.231} C_VEL
LIN {X 0,Y 399.54,Z 796.401,A -85,B 0,C 180,E1 17622.49,E2 17622.49} C_VEL
LIN {X 0,Y 394.468,Z 790.969,A -85,B 0,C 180,E1 17625.659,E2 17625.659} C_VEL
LIN {X 0,Y 393.621,Z 788.459,A -85,B 0,C 180,E1 17626.406,E2 17626.406} C_VEL
LIN {X 0,Y 388.537,Z 783.764,A -85,B 0,C 180,E1 17631.108,E2 17631.108} C_VEL
LIN {X 0,Y 388.013,Z 780.81,A -85,B 0,C 180,E1 17632.305,E2 17632.305} C_VEL
LIN {X 0,Y 388.478,Z 780.81,A -85,B 0,C 180,E1 17637.775,E2 17637.775} C_VEL
LIN {X 0,Y 388.492,Z 780.81,A -85,B 0,C 180,E1 17642.232,E2 17642.232} C_VEL
LIN {X 0,Y 388.202,Z 781.591,A -85,B 0,C 180,E1 17645.657,E2 17645.657} C_VEL
LIN {X 0,Y 391.023,Z 787.007,A -85,B 0,C 180,E1 17649.034,E2 17649.034} C_VEL
LIN {X 0,Y 394.221,Z 789.625,A -85,B 0,C 180,E1 17651.541,E2 17651.541} C_VEL
LIN {X 0,Y 398.051,Z 795.266,A -85,B 0,C 180,E1 17654.146,E2 17654.146} C_VEL
LIN {X 0,Y 400.019,Z 797.357,A -85,B 0,C 180,E1 17655.264,E2 17655.264} C_VEL
LIN {X 0,Y 404.678,Z 803.163,A -85,B 0,C 180,E1 17657.662,E2 17657.662} C_VEL
LIN {X 0,Y 416.614,Z 820.59,A -85,B 0,C 180,E1 17662.807,E2 17662.807} C_VEL
LIN {X 0,Y 428.447,Z 839.043,A -85,B 0,C 180,E1 17667.147,E2 17667.147} C_VEL
LIN {X 0,Y 441.588,Z 863.9,A -85,B 0,C 180,E1 17671.751,E2 17671.751} C_VEL
LIN {X 0,Y 453.435,Z 893.294,A -85,B 0,C 180,E1 17676.188,E2 17676.188} C_VEL
LIN {X 0,Y 459.023,Z 912.271,A -85,B 0,C 180,E1 17678.713,E2 17678.713} C_VEL
LIN {X 0,Y 448.33,Z 952.092,A -85,B 0,C 180,E1 17681.307,E2 17681.307} C_VEL
LIN {X 0,Y 436.441,Z 989.007,A -85,B 0,C 180,E1 17684.609,E2 17684.609} C_VEL
LIN {X 0,Y 424.118,Z 1022.944,A -85,B 0,C 180,E1 17688.718,E2 17688.718} C_VEL
LIN {X 0,Y 411.618,Z 1054.967,A -85,B 0,C 180,E1 17694.03,E2 17694.03} C_VEL
LIN {X 0,Y 401.342,Z 1081.286,A -85,B 0,C 180,E1 17700.098,E2 17700.098} C_VEL
LIN {X 0,Y 394.172,Z 1102.02,A -85,B 0,C 180,E1 17706.921,E2 17706.921} C_VEL
LIN {X 0,Y 390.622,Z 1114.676,A -85,B 0,C 180,E1 17713.135,E2 17713.135} C_VEL
LIN {X 0,Y 389.105,Z 1121.998,A -85,B 0,C 180,E1 17718.805,E2 17718.805} C_VEL
LIN {X 0,Y 388.589,Z 1125.536,A -85,B 0,C 180,E1 17725.541,E2 17725.541} C_VEL
LIN {X 0,Y 388.818,Z 1124.923,A -85,B 0,C 180,E1 17730.001,E2 17730.001} C_VEL
LIN {X 0,Y 389.415,Z 1119.583,A -85,B 0,C 180,E1 17736.686,E2 17736.686} C_VEL
LIN {X 0,Y 391.712,Z 1108.491,A -85,B 0,C 180,E1 17743.384,E2 17743.384} C_VEL
LIN {X 0,Y 395.94,Z 1092.901,A -85,B 0,C 180,E1 17749.51,E2 17749.51} C_VEL
LIN {X 0,Y 402.968,Z 1072.145,A -85,B 0,C 180,E1 17755.347,E2 17755.347} C_VEL
LIN {X 0,Y 413.204,Z 1043.914,A -85,B 0,C 180,E1 17761.103,E2 17761.103} C_VEL
LIN {X 0,Y 424.829,Z 1011.392,A -85,B 0,C 180,E1 17765.939,E2 17765.939} C_VEL
LIN {X 0,Y 436.87,Z 974.61,A -85,B 0,C 180,E1 17769.947,E2 17769.947} C_VEL
LIN {X 0,Y 447.75,Z 935.402,A -85,B 0,C 180,E1 17773.09,E2 17773.09} C_VEL
LIN {X 0,Y 453.831,Z 908.961,A -85,B 0,C 180,E1 17774.724,E2 17774.724} C_VEL
LIN {X 0,Y 443.741,Z 877.253,A -85,B 0,C 180,E1 17778.666,E2 17778.666} C_VEL
LIN {X 0,Y 430.451,Z 847.556,A -85,B 0,C 180,E1 17782.892,E2 17782.892} C_VEL
LIN {X 0,Y 414.506,Z 820.203,A -85,B 0,C 180,E1 17787.707,E2 17787.707} C_VEL
LIN {X 0,Y 401.287,Z 801.354,A -85,B 0,C 180,E1 17791.945,E2 17791.945} C_VEL
LIN {X 0,Y 396.236,Z 794.592,A -85,B 0,C 180,E1 17793.76,E2 17793.76} C_VEL
LIN {X 0,Y 392.441,Z 788.624,A -85,B 0,C 180,E1 17795.287,E2 17795.287} C_VEL
LIN {X 0,Y 387.774,Z 783.967,A -85,B 0,C 180,E1 17797.217,E2 17797.217} C_VEL
LIN {X 0,Y 387.144,Z 780.81,A -85,B 0,C 180,E1 17797.632,E2 17797.632} C_VEL
LIN {X 0,Y 387.493,Z 780.81,A -85,B 0,C 180,E1 17804.158,E2 17804.158} C_VEL
LIN {X 0,Y 387.962,Z 780.81,A -85,B 0,C 180,E1 17811.035,E2 17811.035} C_VEL
LIN {X 0,Y 388.505,Z 780.81,A -85,B 0,C 180,E1 17817.768,E2 17817.768} C_VEL
LIN {X 0,Y 388.502,Z 780.81,A -85,B 0,C 180,E1 17822.225,E2 17822.225} C_VEL
LIN {X 0,Y 387.972,Z 780.81,A -85,B 0,C 180,E1 17828.958,E2 17828.958} C_VEL
LIN {X 0,Y 387.565,Z 780.81,A -85,B 0,C 180,E1 17835.832,E2 17835.832} C_VEL
LIN {X 0,Y 387.337,Z 780.901,A -85,B 0,C 180,E1 17838.916,E2 17838.916} C_VEL
LIN {X 0,Y 388.989,Z 785.679,A -85,B 0,C 180,E1 17839.79,E2 17839.79} C_VEL
LIN {X 0,Y 392.865,Z 789.325,A -85,B 0,C 180,E1 17841.351,E2 17841.351} C_VEL
LIN {X 0,Y 396.984,Z 795.013,A -85,B 0,C 180,E1 17842.954,E2 17842.954} C_VEL
LIN {X 0,Y 412.422,Z 816.625,A -85,B 0,C 180,E1 17848.034,E2 17848.034} C_VEL
LIN {X 0,Y 429.402,Z 843.378,A -85,B 0,C 180,E1 17852.775,E2 17852.775} C_VEL
LIN {X 0,Y 445.548,Z 875.794,A -85,B 0,C 180,E1 17857.231,E2 17857.231} C_VEL
LIN {X 0,Y 457.211,Z 907.733,A -85,B 0,C 180,E1 17860.927,E2 17860.927} C_VEL
LIN {X 0,Y 447.975,Z 950.274,A -85,B 0,C 180,E1 17863.158,E2 17863.158} C_VEL
LIN {X 0,Y 436.544,Z 991.267,A -85,B 0,C 180,E1 17866.186,E2 17866.186} C_VEL
LIN {X 0,Y 425.043,Z 1027.372,A -85,B 0,C 180,E1 17869.85,E2 17869.85} C_VEL
LIN {X 0,Y 413.977,Z 1059.841,A -85,B 0,C 180,E1 17874.264,E2 17874.264} C_VEL
LIN {X 0,Y 403.999,Z 1088.955,A -85,B 0,C 180,E1 17879.567,E2 17879.567} C_VEL
LIN {X 0,Y 395.884,Z 1114.433,A -85,B 0,C 180,E1 17885.931,E2 17885.931} C_VEL
LIN {X 0,Y 391.199,Z 1133.152,A -85,B 0,C 180,E1 17892.579,E2 17892.579} C_VEL
LIN {X 0,Y 389.171,Z 1144.87,A -85,B 0,C 180,E1 17898.804,E2 17898.804} C_VEL
LIN {X 0,Y 388.786,Z 1150.204,A -85,B 0,C 180,E1 17903.303,E2 17903.303} C_VEL
LIN {X 0,Y 388.745,Z 1152.954,A -85,B 0,C 180,E1 17907.771,E2 17907.771} C_VEL
LIN {X 0,Y 388.708,Z 1153.044,A -85,B 0,C 180,E1 17912.227,E2 17912.227} C_VEL
LIN {X 0,Y 388.865,Z 1149.527,A -85,B 0,C 180,E1 17917.996,E2 17917.996} C_VEL
LIN {X 0,Y 390.076,Z 1140.462,A -85,B 0,C 180,E1 17924.478,E2 17924.478} C_VEL
LIN {X 0,Y 393.289,Z 1126.254,A -85,B 0,C 180,E1 17930.817,E2 17930.817} C_VEL
LIN {X 0,Y 399.513,Z 1106.539,A -85,B 0,C 180,E1 17936.992,E2 17936.992} C_VEL
LIN {X 0,Y 409.099,Z 1079.889,A -85,B 0,C 180,E1 17943.011,E2 17943.011} C_VEL
LIN {X 0,Y 420.976,Z 1048.053,A -85,B 0,C 180,E1 17948.256,E2 17948.256} C_VEL
LIN {X 0,Y 433.374,Z 1013.752,A -85,B 0,C 180,E1 17952.406,E2 17952.406} C_VEL
LIN {X 0,Y 433.085,Z 1005.889,A -85,B 0,C 180,E1 17953.577,E2 17953.577} C_VEL
LIN {X 0,Y 432.643,Z 998.865,A -85,B 0,C 180,E1 17954.599,E2 17954.599} C_VEL
LIN {X 0,Y 432.998,Z 997.711,A -85,B 0,C 180,E1 17954.712,E2 17954.712} C_VEL
LIN {X 0,Y 445.035,Z 959.492,A -85,B 0,C 180,E1 17957.708,E2 17957.708} C_VEL
LIN {X 0,Y 455.735,Z 918.607,A -85,B 0,C 180,E1 17959.998,E2 17959.998} C_VEL
LIN {X 0,Y 456.409,Z 912.513,A -85,B 0,C 180,E1 17960.365,E2 17960.365} C_VEL
LIN {X 0,Y 444.849,Z 881.366,A -85,B 0,C 180,E1 17964.589,E2 17964.589} C_VEL
LIN {X 0,Y 430.619,Z 853.038,A -85,B 0,C 180,E1 17969.351,E2 17969.351} C_VEL
LIN {X 0,Y 416.095,Z 829.735,A -85,B 0,C 180,E1 17974.461,E2 17974.461} C_VEL
LIN {X 0,Y 406.194,Z 816.031,A -85,B 0,C 180,E1 17978.534,E2 17978.534} C_VEL
LIN {X 0,Y 401.392,Z 809.554,A -85,B 0,C 180,E1 17980.845,E2 17980.845} C_VEL
LIN {X 0,Y 396.85,Z 803.162,A -85,B 0,C 180,E1 17983.418,E2 17983.418} C_VEL
LIN {X 0,Y 392.652,Z 797.433,A -85,B 0,C 180,E1 17986.301,E2 17986.301} C_VEL
LIN {X 0,Y 390.911,Z 795.607,A -85,B 0,C 180,E1 17987.681,E2 17987.681} C_VEL
LIN {X 0,Y 387.021,Z 790.253,A -85,B 0,C 180,E1 17991.939,E2 17991.939} C_VEL
LIN {X 0,Y 386.643,Z 788.588,A -85,B 0,C 180,E1 17992.707,E2 17992.707} C_VEL
LIN {X 0,Y 385.805,Z 788.306,A -85,B 0,C 180,E1 18003.371,E2 18003.371} C_VEL
LIN {X 0,Y 387.053,Z 789.602,A -85,B 0,C 180,E1 18005.463,E2 18005.463} C_VEL
LIN {X 0,Y 390.537,Z 795.301,A -85,B 0,C 180,E1 18009.467,E2 18009.467} C_VEL
LIN {X 0,Y 392.783,Z 797.253,A -85,B 0,C 180,E1 18011.232,E2 18011.232} C_VEL
LIN {X 0,Y 396.872,Z 803.056,A -85,B 0,C 180,E1 18014.049,E2 18014.049} C_VEL
LIN {X 0,Y 398.771,Z 805.725,A -85,B 0,C 180,E1 18015.179,E2 18015.179} C_VEL
LIN {X 0,Y 404.159,Z 813.153,A -85,B 0,C 180,E1 18018.037,E2 18018.037} C_VEL
LIN {X 0,Y 413.38,Z 826.421,A -85,B 0,C 180,E1 18022.146,E2 18022.146} C_VEL
LIN {X 0,Y 425.23,Z 845.765,A -85,B 0,C 180,E1 18026.798,E2 18026.798} C_VEL
LIN {X 0,Y 437.202,Z 869.199,A -85,B 0,C 180,E1 18031.226,E2 18031.226} C_VEL
LIN {X 0,Y 448.795,Z 899.461,A -85,B 0,C 180,E1 18035.912,E2 18035.912} C_VEL
LIN {X 0,Y 453.017,Z 916.257,A -85,B 0,C 180,E1 18038.157,E2 18038.157} C_VEL
LIN {X 0,Y 441.445,Z 957.274,A -85,B 0,C 180,E1 18040.927,E2 18040.927} C_VEL
LIN {X 0,Y 428.284,Z 995.903,A -85,B 0,C 180,E1 18044.582,E2 18044.582} C_VEL
LIN {X 0,Y 415.585,Z 1029.094,A -85,B 0,C 180,E1 18048.893,E2 18048.893} C_VEL
LIN {X 0,Y 404.426,Z 1056.408,A -85,B 0,C 180,E1 18053.62,E2 18053.62} C_VEL
LIN {X 0,Y 394.005,Z 1082.093,A -85,B 0,C 180,E1 18059.686,E2 18059.686} C_VEL
LIN {X 0,Y 386.642,Z 1102.21,A -85,B 0,C 180,E1 18066.445,E2 18066.445} C_VEL
LIN {X 0,Y 382.898,Z 1114.9,A -85,B 0,C 180,E1 18072.785,E2 18072.785} C_VEL
LIN {X 0,Y 381.248,Z 1122.242,A -85,B 0,C 180,E1 18078.571,E2 18078.571} C_VEL
LIN {X 0,Y 380.683,Z 1125.812,A -85,B 0,C 180,E1 18085.448,E2 18085.448} C_VEL
LIN {X 0,Y 380.92,Z 1125.221,A -85,B 0,C 180,E1 18090.001,E2 18090.001} C_VEL
LIN {X 0,Y 381.552,Z 1119.916,A -85,B 0,C 180,E1 18096.825,E2 18096.825} C_VEL
LIN {X 0,Y 383.961,Z 1108.849,A -85,B 0,C 180,E1 18103.66,E2 18103.66} C_VEL
LIN {X 0,Y 388.417,Z 1093.298,A -85,B 0,C 180,E1 18109.903,E2 18109.903} C_VEL
LIN {X 0,Y 395.594,Z 1073.057,A -85,B 0,C 180,E1 18115.731,E2 18115.731} C_VEL
LIN {X 0,Y 406.407,Z 1044.4,A -85,B 0,C 180,E1 18121.683,E2 18121.683} C_VEL
LIN {X 0,Y 418.418,Z 1011.918,A -85,B 0,C 180,E1 18126.578,E2 18126.578} C_VEL
LIN {X 0,Y 430.742,Z 975.448,A -85,B 0,C 180,E1 18130.601,E2 18130.601} C_VEL
LIN {X 0,Y 441.767,Z 937.09,A -85,B 0,C 180,E1 18133.721,E2 18133.721} C_VEL
LIN {X 0,Y 447.663,Z 911.466,A -85,B 0,C 180,E1 18135.375,E2 18135.375} C_VEL
LIN {X 0,Y 438.059,Z 880.409,A -85,B 0,C 180,E1 18139.369,E2 18139.369} C_VEL
LIN {X 0,Y 425.392,Z 851.548,A -85,B 0,C 180,E1 18143.649,E2 18143.649} C_VEL
LIN {X 0,Y 410.587,Z 825.681,A -85,B 0,C 180,E1 18148.372,E2 18148.372} C_VEL
LIN {X 0,Y 398.21,Z 807.562,A -85,B 0,C 180,E1 18152.594,E2 18152.594} C_VEL
LIN {X 0,Y 393.698,Z 801.437,A -85,B 0,C 180,E1 18154.284,E2 18154.284} C_VEL
LIN {X 0,Y 388.949,Z 794.968,A -85,B 0,C 180,E1 18156.23,E2 18156.23} C_VEL
LIN {X 0,Y 385.154,Z 789.5,A -85,B 0,C 180,E1 18157.965,E2 18157.965} C_VEL
LIN {X 0,Y 379.699,Z 783.127,A -85,B 0,C 180,E1 18160.726,E2 18160.726} C_VEL
LIN {X 0,Y 379.375,Z 780.81,A -85,B 0,C 180,E1 18161.135,E2 18161.135} C_VEL
LIN {X 0,Y 379.888,Z 780.81,A -85,B 0,C 180,E1 18168.526,E2 18168.526} C_VEL
LIN {X 0,Y 380.383,Z 780.81,A -85,B 0,C 180,E1 18175.44,E2 18175.44} C_VEL
LIN {X 0,Y 380.772,Z 780.81,A -85,B 0,C 180,E1 18179.997,E2 18179.997} C_VEL
LIN {X 0,Y 380.219,Z 780.81,A -85,B 0,C 180,E1 18186.843,E2 18186.843} C_VEL
LIN {X 0,Y 379.749,Z 780.81,A -85,B 0,C 180,E1 18193.807,E2 18193.807} C_VEL
LIN {X 0,Y 379.661,Z 780.924,A -85,B 0,C 180,E1 18195.578,E2 18195.578} C_VEL
LIN {X 0,Y 381.423,Z 785.923,A -85,B 0,C 180,E1 18196.703,E2 18196.703} C_VEL
LIN {X 0,Y 385.311,Z 789.5,A -85,B 0,C 180,E1 18198.558,E2 18198.558} C_VEL
LIN {X 0,Y 389.476,Z 795.147,A -85,B 0,C 180,E1 18200.43,E2 18200.43} C_VEL
LIN {X 0,Y 401.221,Z 811.439,A -85,B 0,C 180,E1 18204.894,E2 18204.894} C_VEL
LIN {X 0,Y 416.92,Z 834.491,A -85,B 0,C 180,E1 18209.775,E2 18209.775} C_VEL
LIN {X 0,Y 432.626,Z 863.009,A -85,B 0,C 180,E1 18214.344,E2 18214.344} C_VEL
LIN {X 0,Y 445.367,Z 892.925,A -85,B 0,C 180,E1 18218.248,E2 18218.248} C_VEL
LIN {X 0,Y 451.212,Z 911.607,A -85,B 0,C 180,E1 18220.389,E2 18220.389} C_VEL
LIN {X 0,Y 442.013,Z 951.482,A -85,B 0,C 180,E1 18222.509,E2 18222.509} C_VEL
LIN {X 0,Y 429.832,Z 993.592,A -85,B 0,C 180,E1 18225.683,E2 18225.683} C_VEL
LIN {X 0,Y 416.98,Z 1032.408,A -85,B 0,C 180,E1 18229.794,E2 18229.794} C_VEL
LIN {X 0,Y 405.069,Z 1065.73,A -85,B 0,C 180,E1 18234.635,E2 18234.635} C_VEL
LIN {X 0,Y 395.528,Z 1092.301,A -85,B 0,C 180,E1 18239.809,E2 18239.809} C_VEL
LIN {X 0,Y 387.889,Z 1115.853,A -85,B 0,C 180,E1 18246.001,E2 18246.001} C_VEL
LIN {X 0,Y 383.197,Z 1134.153,A -85,B 0,C 180,E1 18252.796,E2 18252.796} C_VEL
LIN {X 0,Y 381.147,Z 1146.159,A -85,B 0,C 180,E1 18259.722,E2 18259.722} C_VEL
LIN {X 0,Y 380.778,Z 1151.606,A -85,B 0,C 180,E1 18265.446,E2 18265.446} C_VEL
LIN {X 0,Y 380.96,Z 1153.034,A -85,B 0,C 180,E1 18269.999,E2 18269.999} C_VEL
LIN {X 0,Y 380.886,Z 1150.368,A -85,B 0,C 180,E1 18276.834,E2 18276.834} C_VEL
LIN {X 0,Y 381.613,Z 1143.836,A -85,B 0,C 180,E1 18282.578,E2 18282.578} C_VEL
LIN {X 0,Y 384.129,Z 1131.892,A -85,B 0,C 180,E1 18288.873,E2 18288.873} C_VEL
LIN {X 0,Y 389.404,Z 1114.255,A -85,B 0,C 180,E1 18295.267,E2 18295.267} C_VEL
LIN {X 0,Y 398.39,Z 1089.612,A -85,B 0,C 180,E1 18301.604,E2 18301.604} C_VEL
LIN {X 0,Y 410.118,Z 1059.621,A -85,B 0,C 180,E1 18307.186,E2 18307.186} C_VEL
LIN {X 0,Y 422.619,Z 1026.895,A -85,B 0,C 180,E1 18311.667,E2 18311.667} C_VEL
LIN {X 0,Y 432.998,Z 997.711,A -85,B 0,C 180,E1 18314.712,E2 18314.712} C_VEL
LIN {X 0,Y 434.816,Z 984.527,A -85,B 0,C 180,E1 18316.214,E2 18316.214} C_VEL
LIN {X 0,Y 436.236,Z 970.956,A -85,B 0,C 180,E1 18317.672,E2 18317.672} C_VEL
LIN {X 0,Y 447.329,Z 932.195,A -85,B 0,C 180,E1 18320.106,E2 18320.106} C_VEL
LIN {X 0,Y 450.86,Z 916.114,A -85,B 0,C 180,E1 18320.954,E2 18320.954} C_VEL
LIN {X 0,Y 439.984,Z 885.776,A -85,B 0,C 180,E1 18325.22,E2 18325.22} C_VEL
LIN {X 0,Y 426.495,Z 858.387,A -85,B 0,C 180,E1 18329.98,E2 18329.98} C_VEL
LIN {X 0,Y 413.235,Z 836.252,A -85,B 0,C 180,E1 18334.996,E2 18334.996} C_VEL
LIN {X 0,Y 404.092,Z 823.232,A -85,B 0,C 180,E1 18338.926,E2 18338.926} C_VEL
LIN {X 0,Y 399.544,Z 816.752,A -85,B 0,C 180,E1 18341.255,E2 18341.255} C_VEL
LIN {X 0,Y 395.156,Z 810.576,A -85,B 0,C 180,E1 18343.818,E2 18343.818} C_VEL
LIN {X 0,Y 391.067,Z 804.466,A -85,B 0,C 180,E1 18346.773,E2 18346.773} C_VEL
LIN {X 0,Y 385.95,Z 798.147,A -85,B 0,C 180,E1 18352.058,E2 18352.058} C_VEL
LIN {X 0,Y 385.318,Z 796.339,A -85,B 0,C 180,E1 18353.248,E2 18353.248} C_VEL
LIN {X 0,Y 384.845,Z 796.135,A -85,B 0,C 180,E1 18363.379,E2 18363.379} C_VEL
LIN {X 0,Y 385.932,Z 797.43,A -85,B 0,C 180,E1 18365.268,E2 18365.268} C_VEL
LIN {X 0,Y 389.585,Z 803.154,A -85,B 0,C 180,E1 18369.49,E2 18369.49} C_VEL
LIN {X 0,Y 391.436,Z 805.059,A -85,B 0,C 180,E1 18370.99,E2 18370.99} C_VEL
LIN {X 0,Y 396.011,Z 811.062,A -85,B 0,C 180,E1 18374.165,E2 18374.165} C_VEL
LIN {X 0,Y 406.123,Z 826.017,A -85,B 0,C 180,E1 18379.617,E2 18379.617} C_VEL
LIN {X 0,Y 418.027,Z 845.264,A -85,B 0,C 180,E1 18384.837,E2 18384.837} C_VEL
LIN {X 0,Y 430.342,Z 868.98,A -85,B 0,C 180,E1 18389.733,E2 18389.733} C_VEL
LIN {X 0,Y 441.369,Z 897.067,A -85,B 0,C 180,E1 18394.394,E2 18394.394} C_VEL
LIN {X 0,Y 447.285,Z 918.323,A -85,B 0,C 180,E1 18397.449,E2 18397.449} C_VEL
LIN {X 0,Y 435.643,Z 958.941,A -85,B 0,C 180,E1 18400.263,E2 18400.263} C_VEL
LIN {X 0,Y 421.778,Z 998.198,A -85,B 0,C 180,E1 18404.048,E2 18404.048} C_VEL
LIN {X 0,Y 408.038,Z 1032.626,A -85,B 0,C 180,E1 18408.667,E2 18408.667} C_VEL
LIN {X 0,Y 395.923,Z 1061.029,A -85,B 0,C 180,E1 18413.875,E2 18413.875} C_VEL
LIN {X 0,Y 386.41,Z 1083.496,A -85,B 0,C 180,E1 18419.445,E2 18419.445} C_VEL
LIN {X 0,Y 379.21,Z 1102.252,A -85,B 0,C 180,E1 18425.894,E2 18425.894} C_VEL
LIN {X 0,Y 375.166,Z 1115.125,A -85,B 0,C 180,E1 18432.418,E2 18432.418} C_VEL
LIN {X 0,Y 373.395,Z 1122.488,A -85,B 0,C 180,E1 18438.327,E2 18438.327} C_VEL
LIN {X 0,Y 372.78,Z 1126.088,A -85,B 0,C 180,E1 18445.351,E2 18445.351} C_VEL
LIN {X 0,Y 373.044,Z 1125.518,A -85,B 0,C 180,E1 18450.001,E2 18450.001} C_VEL
LIN {X 0,Y 373.714,Z 1120.245,A -85,B 0,C 180,E1 18456.969,E2 18456.969} C_VEL
LIN {X 0,Y 376.244,Z 1109.206,A -85,B 0,C 180,E1 18463.946,E2 18463.946} C_VEL
LIN {X 0,Y 380.918,Z 1093.694,A -85,B 0,C 180,E1 18470.312,E2 18470.312} C_VEL
LIN {X 0,Y 388.82,Z 1072.347,A -85,B 0,C 180,E1 18476.518,E2 18476.518} C_VEL
LIN {X 0,Y 399.644,Z 1044.884,A -85,B 0,C 180,E1 18482.283,E2 18482.283} C_VEL
LIN {X 0,Y 412.052,Z 1012.443,A -85,B 0,C 180,E1 18487.237,E2 18487.237} C_VEL
LIN {X 0,Y 424.27,Z 977.49,A -85,B 0,C 180,E1 18491.157,E2 18491.157} C_VEL
LIN {X 0,Y 435.56,Z 939.833,A -85,B 0,C 180,E1 18494.294,E2 18494.294} C_VEL
LIN {X 0,Y 441.81,Z 915.007,A -85,B 0,C 180,E1 18495.912,E2 18495.912} C_VEL
LIN {X 0,Y 432.843,Z 884.709,A -85,B 0,C 180,E1 18499.934,E2 18499.934} C_VEL
LIN {X 0,Y 420.52,Z 855.817,A -85,B 0,C 180,E1 18504.355,E2 18504.355} C_VEL
LIN {X 0,Y 405.514,Z 828.848,A -85,B 0,C 180,E1 18509.478,E2 18509.478} C_VEL
LIN {X 0,Y 392.098,Z 809.122,A -85,B 0,C 180,E1 18514.452,E2 18514.452} C_VEL
LIN {X 0,Y 386.307,Z 801.708,A -85,B 0,C 180,E1 18516.884,E2 18516.884} C_VEL
LIN {X 0,Y 381.934,Z 795.391,A -85,B 0,C 180,E1 18518.989,E2 18518.989} C_VEL
LIN {X 0,Y 377.732,Z 789.962,A -85,B 0,C 180,E1 18521.259,E2 18521.259} C_VEL
LIN {X 0,Y 376.489,Z 788.136,A -85,B 0,C 180,E1 18522.014,E2 18522.014} C_VEL
LIN {X 0,Y 372.101,Z 783.415,A -85,B 0,C 180,E1 18524.92,E2 18524.92} C_VEL
LIN {X 0,Y 371.722,Z 780.81,A -85,B 0,C 180,E1 18525.581,E2 18525.581} C_VEL
LIN {X 0,Y 372.28,Z 780.81,A -85,B 0,C 180,E1 18533.277,E2 18533.277} C_VEL
LIN {X 0,Y 372.875,Z 780.81,A -85,B 0,C 180,E1 18539.996,E2 18539.996} C_VEL
LIN {X 0,Y 372.288,Z 780.81,A -85,B 0,C 180,E1 18546.989,E2 18546.989} C_VEL
LIN {X 0,Y 372.05,Z 781.413,A -85,B 0,C 180,E1 18551.34,E2 18551.34} C_VEL
LIN {X 0,Y 373.932,Z 786.163,A -85,B 0,C 180,E1 18552.888,E2 18552.888} C_VEL
LIN {X 0,Y 377.834,Z 789.302,A -85,B 0,C 180,E1 18555.21,E2 18555.21} C_VEL
LIN {X 0,Y 381.193,Z 794.769,A -85,B 0,C 180,E1 18557.112,E2 18557.112} C_VEL
LIN {X 0,Y 383.567,Z 797.361,A -85,B 0,C 180,E1 18558.267,E2 18558.267} C_VEL
LIN {X 0,Y 389.657,Z 805.909,A -85,B 0,C 180,E1 18561.005,E2 18561.005} C_VEL
LIN {X 0,Y 398.931,Z 818.58,A -85,B 0,C 180,E1 18564.517,E2 18564.517} C_VEL
LIN {X 0,Y 413.574,Z 840.874,A -85,B 0,C 180,E1 18569.32,E2 18569.32} C_VEL
LIN {X 0,Y 427.843,Z 867.564,A -85,B 0,C 180,E1 18573.712,E2 18573.712} C_VEL
LIN {X 0,Y 440.157,Z 897.539,A -85,B 0,C 180,E1 18577.759,E2 18577.759} C_VEL
LIN {X 0,Y 445.315,Z 914.221,A -85,B 0,C 180,E1 18579.751,E2 18579.751} C_VEL
LIN {X 0,Y 435.646,Z 954.314,A -85,B 0,C 180,E1 18581.96,E2 18581.96} C_VEL
LIN {X 0,Y 423.691,Z 994.257,A -85,B 0,C 180,E1 18585.026,E2 18585.026} C_VEL
LIN {X 0,Y 410.159,Z 1033.646,A -85,B 0,C 180,E1 18589.27,E2 18589.27} C_VEL
LIN {X 0,Y 397.153,Z 1068.702,A -85,B 0,C 180,E1 18594.531,E2 18594.531} C_VEL
LIN {X 0,Y 386.574,Z 1097.175,A -85,B 0,C 180,E1 18600.427,E2 18600.427} C_VEL
LIN {X 0,Y 378.933,Z 1120.389,A -85,B 0,C 180,E1 18607.118,E2 18607.118} C_VEL
LIN {X 0,Y 374.894,Z 1136.172,A -85,B 0,C 180,E1 18613.61,E2 18613.61} C_VEL
LIN {X 0,Y 373.282,Z 1145.839,A -85,B 0,C 180,E1 18619.503,E2 18619.503} C_VEL
LIN {X 0,Y 372.875,Z 1151.313,A -85,B 0,C 180,E1 18625.35,E2 18625.35} C_VEL
LIN {X 0,Y 373.08,Z 1152.75,A -85,B 0,C 180,E1 18629.999,E2 18629.999} C_VEL
LIN {X 0,Y 373.001,Z 1150.104,A -85,B 0,C 180,E1 18636.979,E2 18636.979} C_VEL
LIN {X 0,Y 373.789,Z 1143.586,A -85,B 0,C 180,E1 18642.846,E2 18642.846} C_VEL
LIN {X 0,Y 376.448,Z 1131.664,A -85,B 0,C 180,E1 18649.273,E2 18649.273} C_VEL
LIN {X 0,Y 382.042,Z 1114.052,A -85,B 0,C 180,E1 18655.789,E2 18655.789} C_VEL
LIN {X 0,Y 391.721,Z 1088.937,A -85,B 0,C 180,E1 18662.341,E2 18662.341} C_VEL
LIN {X 0,Y 403.944,Z 1058.81,A -85,B 0,C 180,E1 18667.996,E2 18667.996} C_VEL
LIN {X 0,Y 416.95,Z 1025.952,A -85,B 0,C 180,E1 18672.508,E2 18672.508} C_VEL
LIN {X 0,Y 429.858,Z 990.513,A -85,B 0,C 180,E1 18676.106,E2 18676.106} C_VEL
LIN {X 0,Y 436.236,Z 970.956,A -85,B 0,C 180,E1 18677.672,E2 18677.672} C_VEL
LIN {X 0,Y 437.763,Z 956.994,A -85,B 0,C 180,E1 18679.061,E2 18679.061} C_VEL
LIN {X 0,Y 439.408,Z 942.572,A -85,B 0,C 180,E1 18680.332,E2 18680.332} C_VEL
LIN {X 0,Y 445.2,Z 919.339,A -85,B 0,C 180,E1 18681.613,E2 18681.613} C_VEL
LIN {X 0,Y 434.9,Z 889.782,A -85,B 0,C 180,E1 18685.907,E2 18685.907} C_VEL
LIN {X 0,Y 421.863,Z 862.582,A -85,B 0,C 180,E1 18690.841,E2 18690.841} C_VEL
LIN {X 0,Y 409.926,Z 842.182,A -85,B 0,C 180,E1 18695.652,E2 18695.652} C_VEL
LIN {X 0,Y 401.238,Z 829.333,A -85,B 0,C 180,E1 18699.692,E2 18699.692} C_VEL
LIN {X 0,Y 397.224,Z 823.623,A -85,B 0,C 180,E1 18701.841,E2 18701.841} C_VEL
LIN {X 0,Y 393.398,Z 817.961,A -85,B 0,C 180,E1 18704.243,E2 18704.243} C_VEL
LIN {X 0,Y 388.782,Z 811.253,A -85,B 0,C 180,E1 18707.811,E2 18707.811} C_VEL
LIN {X 0,Y 384.808,Z 805.757,A -85,B 0,C 180,E1 18712.318,E2 18712.318} C_VEL
LIN {X 0,Y 383.954,Z 804.053,A -85,B 0,C 180,E1 18713.929,E2 18713.929} C_VEL
LIN {X 0,Y 383.883,Z 803.977,A -85,B 0,C 180,E1 18723.388,E2 18723.388} C_VEL
LIN {X 0,Y 384.852,Z 805.386,A -85,B 0,C 180,E1 18725.142,E2 18725.142} C_VEL
LIN {X 0,Y 388.926,Z 811.244,A -85,B 0,C 180,E1 18729.789,E2 18729.789} C_VEL
LIN {X 0,Y 395.389,Z 820.791,A -85,B 0,C 180,E1 18734.606,E2 18734.606} C_VEL
LIN {X 0,Y 400.68,Z 828.822,A -85,B 0,C 180,E1 18737.702,E2 18737.702} C_VEL
LIN {X 0,Y 409.151,Z 842.139,A -85,B 0,C 180,E1 18741.887,E2 18741.887} C_VEL
LIN {X 0,Y 419.971,Z 861.639,A -85,B 0,C 180,E1 18746.653,E2 18746.653} C_VEL
LIN {X 0,Y 431.606,Z 888.22,A -85,B 0,C 180,E1 18751.677,E2 18751.677} C_VEL
LIN {X 0,Y 440.414,Z 916.47,A -85,B 0,C 180,E1 18756.095,E2 18756.095} C_VEL
LIN {X 0,Y 441.227,Z 923.27,A -85,B 0,C 180,E1 18756.962,E2 18756.962} C_VEL
LIN {X 0,Y 429.466,Z 961.672,A -85,B 0,C 180,E1 18759.676,E2 18759.676} C_VEL
LIN {X 0,Y 415.732,Z 999.329,A -85,B 0,C 180,E1 18763.37,E2 18763.37} C_VEL
LIN {X 0,Y 401.48,Z 1033.806,A -85,B 0,C 180,E1 18768.07,E2 18768.07} C_VEL
LIN {X 0,Y 388.676,Z 1062.65,A -85,B 0,C 180,E1 18773.488,E2 18773.488} C_VEL
LIN {X 0,Y 378.482,Z 1085.607,A -85,B 0,C 180,E1 18779.408,E2 18779.408} C_VEL
LIN {X 0,Y 371.261,Z 1103.837,A -85,B 0,C 180,E1 18785.984,E2 18785.984} C_VEL
LIN {X 0,Y 366.918,Z 1117.231,A -85,B 0,C 180,E1 18793.246,E2 18793.246} C_VEL
LIN {X 0,Y 365.572,Z 1122.733,A -85,B 0,C 180,E1 18798.074,E2 18798.074} C_VEL
LIN {X 0,Y 364.875,Z 1126.365,A -85,B 0,C 180,E1 18805.25,E2 18805.25} C_VEL
LIN {X 0,Y 365.146,Z 1125.816,A -85,B 0,C 180,E1 18810.001,E2 18810.001} C_VEL
LIN {X 0,Y 365.855,Z 1120.572,A -85,B 0,C 180,E1 18817.119,E2 18817.119} C_VEL
LIN {X 0,Y 368.521,Z 1109.563,A -85,B 0,C 180,E1 18824.244,E2 18824.244} C_VEL
LIN {X 0,Y 373.438,Z 1094.089,A -85,B 0,C 180,E1 18830.738,E2 18830.738} C_VEL
LIN {X 0,Y 381.667,Z 1072.786,A -85,B 0,C 180,E1 18837.055,E2 18837.055} C_VEL
LIN {X 0,Y 392.914,Z 1045.364,A -85,B 0,C 180,E1 18842.905,E2 18842.905} C_VEL
LIN {X 0,Y 406.449,Z 1011.065,A -85,B 0,C 180,E1 18848.178,E2 18848.178} C_VEL
LIN {X 0,Y 419.973,Z 973.33,A -85,B 0,C 180,E1 18852.338,E2 18852.338} C_VEL
LIN {X 0,Y 432.664,Z 931.016,A -85,B 0,C 180,E1 18855.679,E2 18855.679} C_VEL
LIN {X 0,Y 435.859,Z 918.283,A -85,B 0,C 180,E1 18856.479,E2 18856.479} C_VEL
LIN {X 0,Y 427.538,Z 888.987,A -85,B 0,C 180,E1 18860.495,E2 18860.495} C_VEL
LIN {X 0,Y 415.79,Z 860.57,A -85,B 0,C 180,E1 18865.006,E2 18865.006} C_VEL
LIN {X 0,Y 402.036,Z 834.909,A -85,B 0,C 180,E1 18870.047,E2 18870.047} C_VEL
LIN {X 0,Y 389.577,Z 816.007,A -85,B 0,C 180,E1 18874.935,E2 18874.935} C_VEL
LIN {X 0,Y 383.715,Z 808.277,A -85,B 0,C 180,E1 18877.548,E2 18877.548} C_VEL
LIN {X 0,Y 379.874,Z 802.65,A -85,B 0,C 180,E1 18879.479,E2 18879.479} C_VEL
LIN {X 0,Y 375.742,Z 796.591,A -85,B 0,C 180,E1 18881.839,E2 18881.839} C_VEL
LIN {X 0,Y 370.508,Z 790.548,A -85,B 0,C 180,E1 18885.382,E2 18885.382} C_VEL
LIN {X 0,Y 369.683,Z 788.43,A -85,B 0,C 180,E1 18886.149,E2 18886.149} C_VEL
LIN {X 0,Y 364.679,Z 783.53,A -85,B 0,C 180,E1 18891.434,E2 18891.434} C_VEL
LIN {X 0,Y 364.355,Z 780.81,A -85,B 0,C 180,E1 18892.85,E2 18892.85} C_VEL
LIN {X 0,Y 364.972,Z 780.81,A -85,B 0,C 180,E1 18899.996,E2 18899.996} C_VEL
LIN {X 0,Y 364.571,Z 781.464,A -85,B 0,C 180,E1 18904.527,E2 18904.527} C_VEL
LIN {X 0,Y 366.599,Z 786.353,A -85,B 0,C 180,E1 18907.545,E2 18907.545} C_VEL
LIN {X 0,Y 370.543,Z 789.539,A -85,B 0,C 180,E1 18911.015,E2 18911.015} C_VEL
LIN {X 0,Y 373.671,Z 794.797,A -85,B 0,C 180,E1 18913.371,E2 18913.371} C_VEL
LIN {X 0,Y 376.22,Z 797.157,A -85,B 0,C 180,E1 18914.904,E2 18914.904} C_VEL
LIN {X 0,Y 380.441,Z 802.885,A -85,B 0,C 180,E1 18917.245,E2 18917.245} C_VEL
LIN {X 0,Y 388.302,Z 814.124,A -85,B 0,C 180,E1 18920.912,E2 18920.912} C_VEL
LIN {X 0,Y 400.161,Z 831.023,A -85,B 0,C 180,E1 18925.446,E2 18925.446} C_VEL
LIN {X 0,Y 414.766,Z 855.388,A -85,B 0,C 180,E1 18930.355,E2 18930.355} C_VEL
LIN {X 0,Y 428.302,Z 884.23,A -85,B 0,C 180,E1 18934.853,E2 18934.853} C_VEL
LIN {X 0,Y 439.48,Z 916.774,A -85,B 0,C 180,E1 18939.092,E2 18939.092} C_VEL
LIN {X 0,Y 429.273,Z 957.135,A -85,B 0,C 180,E1 18941.388,E2 18941.388} C_VEL
LIN {X 0,Y 416.985,Z 996.491,A -85,B 0,C 180,E1 18944.498,E2 18944.498} C_VEL
LIN {X 0,Y 404.017,Z 1033.059,A -85,B 0,C 180,E1 18948.499,E2 18948.499} C_VEL
LIN {X 0,Y 390.525,Z 1068.267,A -85,B 0,C 180,E1 18953.835,E2 18953.835} C_VEL
LIN {X 0,Y 379.507,Z 1096.77,A -85,B 0,C 180,E1 18959.82,E2 18959.82} C_VEL
LIN {X 0,Y 371.414,Z 1120.016,A -85,B 0,C 180,E1 18966.628,E2 18966.628} C_VEL
LIN {X 0,Y 367.146,Z 1135.832,A -85,B 0,C 180,E1 18973.254,E2 18973.254} C_VEL
LIN {X 0,Y 365.409,Z 1145.519,A -85,B 0,C 180,E1 18979.274,E2 18979.274} C_VEL
LIN {X 0,Y 364.971,Z 1151.019,A -85,B 0,C 180,E1 18985.249,E2 18985.249} C_VEL
LIN {X 0,Y 365.182,Z 1152.464,A -85,B 0,C 180,E1 18989.999,E2 18989.999} C_VEL
LIN {X 0,Y 365.126,Z 1149.841,A -85,B 0,C 180,E1 18997.131,E2 18997.131} C_VEL
LIN {X 0,Y 365.952,Z 1143.335,A -85,B 0,C 180,E1 19003.125,E2 19003.125} C_VEL
LIN {X 0,Y 368.85,Z 1131.069,A -85,B 0,C 180,E1 19009.854,E2 19009.854} C_VEL
LIN {X 0,Y 374.726,Z 1113.85,A -85,B 0,C 180,E1 19016.331,E2 19016.331} C_VEL
LIN {X 0,Y 384.828,Z 1088.76,A -85,B 0,C 180,E1 19022.993,E2 19022.993} C_VEL
LIN {X 0,Y 397.426,Z 1058.961,A -85,B 0,C 180,E1 19028.672,E2 19028.672} C_VEL
LIN {X 0,Y 410.632,Z 1026.827,A -85,B 0,C 180,E1 19033.156,E2 19033.156} C_VEL
LIN {X 0,Y 423.855,Z 991.888,A -85,B 0,C 180,E1 19036.77,E2 19036.77} C_VEL
LIN {X 0,Y 437.405,Z 949.961,A -85,B 0,C 180,E1 19039.893,E2 19039.893} C_VEL
LIN {X 0,Y 439.408,Z 942.572,A -85,B 0,C 180,E1 19040.332,E2 19040.332} C_VEL
LIN {X 0,Y 440.204,Z 932.872,A -85,B 0,C 180,E1 19041.183,E2 19041.183} C_VEL
LIN {X 0,Y 439.491,Z 923.56,A -85,B 0,C 180,E1 19042.177,E2 19042.177} C_VEL
LIN {X 0,Y 431.464,Z 898.002,A -85,B 0,C 180,E1 19045.929,E2 19045.929} C_VEL
LIN {X 0,Y 419.659,Z 871.438,A -85,B 0,C 180,E1 19050.75,E2 19050.75} C_VEL
LIN {X 0,Y 407.828,Z 849.886,A -85,B 0,C 180,E1 19055.81,E2 19055.81} C_VEL
LIN {X 0,Y 396.926,Z 832.588,A -85,B 0,C 180,E1 19061.342,E2 19061.342} C_VEL
LIN {X 0,Y 391.614,Z 825.374,A -85,B 0,C 180,E1 19064.622,E2 19064.622} C_VEL
LIN {X 0,Y 387.291,Z 818.811,A -85,B 0,C 180,E1 19068.161,E2 19068.161} C_VEL
LIN {X 0,Y 383.606,Z 813.107,A -85,B 0,C 180,E1 19072.72,E2 19072.72} C_VEL
LIN {X 0,Y 382.608,Z 811.776,A -85,B 0,C 180,E1 19074.691,E2 19074.691} C_VEL
LIN {X 0,Y 383.509,Z 812.049,A -85,B 0,C 180,E1 19084.452,E2 19084.452} C_VEL
LIN {X 0,Y 386.728,Z 818.361,A -85,B 0,C 180,E1 19088.888,E2 19088.888} C_VEL
LIN {X 0,Y 388.676,Z 820.838,A -85,B 0,C 180,E1 19090.644,E2 19090.644} C_VEL
LIN {X 0,Y 393.726,Z 828.626,A -85,B 0,C 180,E1 19094.458,E2 19094.458} C_VEL
LIN {X 0,Y 401.276,Z 840.173,A -85,B 0,C 180,E1 19098.882,E2 19098.882} C_VEL
LIN {X 0,Y 411.993,Z 859.376,A -85,B 0,C 180,E1 19104.246,E2 19104.246} C_VEL
LIN {X 0,Y 422.635,Z 882.311,A -85,B 0,C 180,E1 19109.152,E2 19109.152} C_VEL
LIN {X 0,Y 431.826,Z 908.762,A -85,B 0,C 180,E1 19113.743,E2 19113.743} C_VEL
LIN {X 0,Y 435.644,Z 925.883,A -85,B 0,C 180,E1 19116.284,E2 19116.284} C_VEL
LIN {X 0,Y 423.844,Z 963.002,A -85,B 0,C 180,E1 19118.954,E2 19118.954} C_VEL
LIN {X 0,Y 409.72,Z 1000.471,A -85,B 0,C 180,E1 19122.679,E2 19122.679} C_VEL
LIN {X 0,Y 395.396,Z 1033.93,A -85,B 0,C 180,E1 19127.286,E2 19127.286} C_VEL
LIN {X 0,Y 382.172,Z 1062.527,A -85,B 0,C 180,E1 19132.697,E2 19132.697} C_VEL
LIN {X 0,Y 371.66,Z 1085.309,A -85,B 0,C 180,E1 19138.621,E2 19138.621} C_VEL
LIN {X 0,Y 363.775,Z 1104.042,A -85,B 0,C 180,E1 19145.457,E2 19145.457} C_VEL
LIN {X 0,Y 359.176,Z 1117.456,A -85,B 0,C 180,E1 19152.874,E2 19152.874} C_VEL
LIN {X 0,Y 357.724,Z 1122.979,A -85,B 0,C 180,E1 19157.808,E2 19157.808} C_VEL
LIN {X 0,Y 356.982,Z 1126.641,A -85,B 0,C 180,E1 19165.145,E2 19165.145} C_VEL
LIN {X 0,Y 357.271,Z 1126.112,A -85,B 0,C 180,E1 19170.001,E2 19170.001} C_VEL
LIN {X 0,Y 358.003,Z 1120.897,A -85,B 0,C 180,E1 19177.276,E2 19177.276} C_VEL
LIN {X 0,Y 360.814,Z 1109.92,A -85,B 0,C 180,E1 19184.555,E2 19184.555} C_VEL
LIN {X 0,Y 365.983,Z 1094.484,A -85,B 0,C 180,E1 19191.18,E2 19191.18} C_VEL
LIN {X 0,Y 374.395,Z 1073.678,A -85,B 0,C 180,E1 19197.498,E2 19197.498} C_VEL
LIN {X 0,Y 386.237,Z 1045.837,A -85,B 0,C 180,E1 19203.549,E2 19203.549} C_VEL
LIN {X 0,Y 400.238,Z 1011.602,A -85,B 0,C 180,E1 19208.881,E2 19208.881} C_VEL
LIN {X 0,Y 414.408,Z 973.266,A -85,B 0,C 180,E1 19213.137,E2 19213.137} C_VEL
LIN {X 0,Y 427.207,Z 931.712,A -85,B 0,C 180,E1 19216.433,E2 19216.433} C_VEL
LIN {X 0,Y 429.865,Z 921.164,A -85,B 0,C 180,E1 19217.116,E2 19217.116} C_VEL
LIN {X 0,Y 421.616,Z 891.325,A -85,B 0,C 180,E1 19221.365,E2 19221.365} C_VEL
LIN {X 0,Y 410.265,Z 863.393,A -85,B 0,C 180,E1 19226.008,E2 19226.008} C_VEL
LIN {X 0,Y 397.541,Z 839.422,A -85,B 0,C 180,E1 19231.008,E2 19231.008} C_VEL
LIN {X 0,Y 386.848,Z 822.624,A -85,B 0,C 180,E1 19235.523,E2 19235.523} C_VEL
LIN {X 0,Y 377.935,Z 809.931,A -85,B 0,C 180,E1 19239.91,E2 19239.91} C_VEL
LIN {X 0,Y 372.925,Z 803.064,A -85,B 0,C 180,E1 19242.915,E2 19242.915} C_VEL
LIN {X 0,Y 368.866,Z 797.448,A -85,B 0,C 180,E1 19245.921,E2 19245.921} C_VEL
LIN {X 0,Y 367.359,Z 795.738,A -85,B 0,C 180,E1 19247.225,E2 19247.225} C_VEL
LIN {X 0,Y 363.29,Z 790.195,A -85,B 0,C 180,E1 19252.228,E2 19252.228} C_VEL
LIN {X 0,Y 362.705,Z 788.532,A -85,B 0,C 180,E1 19253.569,E2 19253.569} C_VEL
LIN {X 0,Y 363.364,Z 788.867,A -85,B 0,C 180,E1 19264.094,E2 19264.094} C_VEL
LIN {X 0,Y 365.497,Z 794.153,A -85,B 0,C 180,E1 19267.418,E2 19267.418} C_VEL
LIN {X 0,Y 369.091,Z 797.22,A -85,B 0,C 180,E1 19270.678,E2 19270.678} C_VEL
LIN {X 0,Y 372.722,Z 802.731,A -85,B 0,C 180,E1 19273.406,E2 19273.406} C_VEL
LIN {X 0,Y 374.844,Z 805.341,A -85,B 0,C 180,E1 19274.736,E2 19274.736} C_VEL
LIN {X 0,Y 380.632,Z 813.499,A -85,B 0,C 180,E1 19277.921,E2 19277.921} C_VEL
LIN {X 0,Y 389.087,Z 825.13,A -85,B 0,C 180,E1 19281.759,E2 19281.759} C_VEL
LIN {X 0,Y 403.434,Z 847.625,A -85,B 0,C 180,E1 19287.228,E2 19287.228} C_VEL
LIN {X 0,Y 417.399,Z 874.762,A -85,B 0,C 180,E1 19292.142,E2 19292.142} C_VEL
LIN {X 0,Y 429.219,Z 905.054,A -85,B 0,C 180,E1 19296.54,E2 19296.54} C_VEL
LIN {X 0,Y 433.456,Z 920.652,A -85,B 0,C 180,E1 19298.495,E2 19298.495} C_VEL
LIN {X 0,Y 422.001,Z 963.413,A -85,B 0,C 180,E1 19301.042,E2 19301.042} C_VEL
LIN {X 0,Y 408.937,Z 1002.841,A -85,B 0,C 180,E1 19304.365,E2 19304.365} C_VEL
LIN {X 0,Y 396.273,Z 1036.798,A -85,B 0,C 180,E1 19308.291,E2 19308.291} C_VEL
LIN {X 0,Y 383.309,Z 1069.324,A -85,B 0,C 180,E1 19313.395,E2 19313.395} C_VEL
LIN {X 0,Y 371.978,Z 1097.564,A -85,B 0,C 180,E1 19319.482,E2 19319.482} C_VEL
LIN {X 0,Y 363.696,Z 1120.415,A -85,B 0,C 180,E1 19326.383,E2 19326.383} C_VEL
LIN {X 0,Y 359.113,Z 1136.669,A -85,B 0,C 180,E1 19333.498,E2 19333.498} C_VEL
LIN {X 0,Y 357.402,Z 1146.62,A -85,B 0,C 180,E1 19340.262,E2 19340.262} C_VEL
LIN {X 0,Y 357.076,Z 1150.726,A -85,B 0,C 180,E1 19345.143,E2 19345.143} C_VEL
LIN {X 0,Y 357.305,Z 1152.18,A -85,B 0,C 180,E1 19349.999,E2 19349.999} C_VEL
LIN {X 0,Y 357.222,Z 1149.577,A -85,B 0,C 180,E1 19357.289,E2 19357.289} C_VEL
LIN {X 0,Y 358.364,Z 1142.056,A -85,B 0,C 180,E1 19364.163,E2 19364.163} C_VEL
LIN {X 0,Y 362.068,Z 1128.34,A -85,B 0,C 180,E1 19371.417,E2 19371.417} C_VEL
LIN {X 0,Y 369.143,Z 1109.367,A -85,B 0,C 180,E1 19378.2,E2 19378.2} C_VEL
LIN {X 0,Y 379.085,Z 1086.028,A -85,B 0,C 180,E1 19384.236,E2 19384.236} C_VEL
LIN {X 0,Y 392.298,Z 1056.15,A -85,B 0,C 180,E1 19389.863,E2 19389.863} C_VEL
LIN {X 0,Y 407.68,Z 1019.783,A -85,B 0,C 180,E1 19394.767,E2 19394.767} C_VEL
LIN {X 0,Y 422.267,Z 981.026,A -85,B 0,C 180,E1 19398.488,E2 19398.488} C_VEL
LIN {X 0,Y 434.963,Z 940.617,A -85,B 0,C 180,E1 19401.257,E2 19401.257} C_VEL
LIN {X 0,Y 439.491,Z 923.56,A -85,B 0,C 180,E1 19402.177,E2 19402.177} C_VEL
LIN {X 0,Y 437.318,Z 916.664,A -85,B 0,C 180,E1 19403.204,E2 19403.204} C_VEL
LIN {X 0,Y 427.893,Z 906.219,A -85,B 0,C 180,E1 19405.929,E2 19405.929} C_VEL
LIN {X 0,Y 416.747,Z 879.143,A -85,B 0,C 180,E1 19410.849,E2 19410.849} C_VEL
LIN {X 0,Y 405.047,Z 856.873,A -85,B 0,C 180,E1 19416.145,E2 19416.145} C_VEL
LIN {X 0,Y 394.759,Z 839.891,A -85,B 0,C 180,E1 19421.67,E2 19421.67} C_VEL
LIN {X 0,Y 389.623,Z 832.531,A -85,B 0,C 180,E1 19425.146,E2 19425.146} C_VEL
LIN {X 0,Y 385.802,Z 826.453,A -85,B 0,C 180,E1 19428.444,E2 19428.444} C_VEL
LIN {X 0,Y 382.294,Z 820.577,A -85,B 0,C 180,E1 19433.052,E2 19433.052} C_VEL
LIN {X 0,Y 380.905,Z 819.2,A -85,B 0,C 180,E1 19441.14,E2 19441.14} C_VEL
LIN {X 0,Y 382.428,Z 820.802,A -85,B 0,C 180,E1 19444.748,E2 19444.748} C_VEL
LIN {X 0,Y 386.303,Z 826.742,A -85,B 0,C 180,E1 19449.572,E2 19449.572} C_VEL
LIN {X 0,Y 391.908,Z 836.373,A -85,B 0,C 180,E1 19454.317,E2 19454.317} C_VEL
LIN {X 0,Y 398.795,Z 847.584,A -85,B 0,C 180,E1 19458.644,E2 19458.644} C_VEL
LIN {X 0,Y 408.736,Z 866.197,A -85,B 0,C 180,E1 19463.923,E2 19463.923} C_VEL
LIN {X 0,Y 418.727,Z 889.065,A -85,B 0,C 180,E1 19468.89,E2 19468.89} C_VEL
LIN {X 0,Y 427.239,Z 915.426,A -85,B 0,C 180,E1 19473.546,E2 19473.546} C_VEL
LIN {X 0,Y 429.899,Z 929.25,A -85,B 0,C 180,E1 19475.632,E2 19475.632} C_VEL
LIN {X 0,Y 417.277,Z 967.117,A -85,B 0,C 180,E1 19478.455,E2 19478.455} C_VEL
LIN {X 0,Y 403.174,Z 1002.942,A -85,B 0,C 180,E1 19482.129,E2 19482.129} C_VEL
LIN {X 0,Y 388.644,Z 1035.717,A -85,B 0,C 180,E1 19486.744,E2 19486.744} C_VEL
LIN {X 0,Y 374.128,Z 1066.073,A -85,B 0,C 180,E1 19492.712,E2 19492.712} C_VEL
LIN {X 0,Y 362.439,Z 1090.284,A -85,B 0,C 180,E1 19499.476,E2 19499.476} C_VEL
LIN {X 0,Y 355.023,Z 1107.712,A -85,B 0,C 180,E1 19506.58,E2 19506.58} C_VEL
LIN {X 0,Y 350.978,Z 1119.25,A -85,B 0,C 180,E1 19513.75,E2 19513.75} C_VEL
LIN {X 0,Y 349.437,Z 1125.058,A -85,B 0,C 180,E1 19520.041,E2 19520.041} C_VEL
LIN {X 0,Y 349.08,Z 1126.918,A -85,B 0,C 180,E1 19525.035,E2 19525.035} C_VEL
LIN {X 0,Y 349.372,Z 1126.41,A -85,B 0,C 180,E1 19530.001,E2 19530.001} C_VEL
LIN {X 0,Y 350.174,Z 1121.219,A -85,B 0,C 180,E1 19537.44,E2 19537.44} C_VEL
LIN {X 0,Y 353.107,Z 1110.276,A -85,B 0,C 180,E1 19544.88,E2 19544.88} C_VEL
LIN {X 0,Y 358.544,Z 1094.878,A -85,B 0,C 180,E1 19551.641,E2 19551.641} C_VEL
LIN {X 0,Y 367.613,Z 1073.397,A -85,B 0,C 180,E1 19558.254,E2 19558.254} C_VEL
LIN {X 0,Y 379.625,Z 1046.305,A -85,B 0,C 180,E1 19564.213,E2 19564.213} C_VEL
LIN {X 0,Y 393.732,Z 1012.975,A -85,B 0,C 180,E1 19569.489,E2 19569.489} C_VEL
LIN {X 0,Y 407.458,Z 977.162,A -85,B 0,C 180,E1 19573.569,E2 19573.569} C_VEL
LIN {X 0,Y 419.725,Z 939.37,A -85,B 0,C 180,E1 19576.73,E2 19576.73} C_VEL
LIN {X 0,Y 423.824,Z 923.808,A -85,B 0,C 180,E1 19577.812,E2 19577.812} C_VEL
LIN {X 0,Y 415.955,Z 894.277,A -85,B 0,C 180,E1 19582.171,E2 19582.171} C_VEL
LIN {X 0,Y 405.38,Z 867.594,A -85,B 0,C 180,E1 19586.807,E2 19586.807} C_VEL
LIN {X 0,Y 393.643,Z 844.749,A -85,B 0,C 180,E1 19591.724,E2 19591.724} C_VEL
LIN {X 0,Y 381.394,Z 824.614,A -85,B 0,C 180,E1 19597.443,E2 19597.443} C_VEL
LIN {X 0,Y 375.079,Z 816.311,A -85,B 0,C 180,E1 19600.802,E2 19600.802} C_VEL
LIN {X 0,Y 371.273,Z 810.532,A -85,B 0,C 180,E1 19603.294,E2 19603.294} C_VEL
LIN {X 0,Y 367.326,Z 804.586,A -85,B 0,C 180,E1 19606.392,E2 19606.392} C_VEL
